   Sensorless mode (stCfg.bNoSensors): the TWELVE movement states ignore
   sensor feedback and advance when tStepTimeoutMs expires — the timeout
   doubles as the fixed step duration. Those twelve are both INIT_* sets
   (3), the three RECOVER_* states, both GRIP states and the four Sep/Push
   states. So error codes 1/3/4/5/6/7/8/10/11/12/13/14 are ALL unreachable
   while sensorless — this said "the 4 movement states" and "1/3/4/5",
   which was wrong before the RECOVER chain existed and is wronger now.
   CHECK_PLATE is deliberately NOT covered: it keeps its own
   tPlateWaitTimeoutMs and still needs a plate sensor, so error 9 stays
   reachable. Every bench run so far has had this flag set, which is why no
   movement-timeout path has ever been exercised on a panel. *)
VAR_INPUT
    (* External start pulse (rising-edge; one scan wide). MAIN fires this
       when the robot's CMD:1 arrives via TCP, or a physical PB1 rising
       edge in Auto mode. HMI START button and SimStartAssembly are
       consumed separately below via their own R_TRIGs. *)
    bExtStartPulse        : BOOL;

    (* Global machine-mode gate (GVL_HMI.bAutoMode). While FALSE the cycle is
       held in IDLE: every start trigger is ignored and a running cycle is
       aborted back to IDLE. This is the hard interlock that stops the
       operator or a stray robot edge starting motion while the machine is
       in Manual. *)
    bMachineAuto          : BOOL;

    (* BENCH SOAK FLAG -- log-file testing only. Wired by MAIN from
       GVL_HMI.bTempTestContinuesAutoRun, ticked online from the IDE. No HMI
       control by decision: an operator must not be able to reach it.

       While TRUE -- AND the build is a bench build, see bBenchBuild -- the
       machine self-arms out of NOT_HOMED and starts another bulb every time it
       reaches IDLE, with no operator START, no robot CMD:1 and no sim flag. So
       the log ring and the CSV fill continuously and rotation / retention can
       actually be exercised on a panel.

       LEVEL, not an edge, unlike every other term it is OR-ed into. That is the
       point: it has to re-fire on each arrival in IDLE.

       Three things it deliberately does NOT do, even on a bench build:
         - it does not bypass bMachineAuto, so Manual is still the hard stop;
         - it does not touch ERR, so a fault still ends the run (with bNoSensors
           AND bBypassPlateSensors set, no error code is reachable, so a soak
           should not fault at all -- if it does, that is a real finding);
         - it does not persist. GVL_HMI is plain VAR_GLOBAL, so the FALSE
           initialiser is re-applied on every cold boot and every download.

       NOTHING downstream reads this input directly. It is gated into
       bTempTestRun in Section 0a and every use site reads that. *)
    bTempTestContinuesAutoRun : BOOL;

    (* Per-pair sensor state. MAIN wires each element from stSepSolK/stPushSolK.bIs*. *)
    bSepIsExtended        : ARRAY[1..3] OF BOOL;
    bSepIsRetracted       : ARRAY[1..3] OF BOOL;
    bPushIsExtended       : ARRAY[1..3] OF BOOL;
    bPushIsRetracted      : ARRAY[1..3] OF BOOL;

    (* Grip pistons — L=[1], R=[2]. MAIN wires from stGripSolL/R.bIs*. *)
    bGripIsExtended       : ARRAY[1..2] OF BOOL;
    bGripIsRetracted      : ARRAY[1..2] OF BOOL;

    (* Plate-presence sensors gating CHECK_PLATE. Both must be TRUE before the
       cycle can advance out of CHECK_PLATE into GRIP_EXTENDING. Latched at
       cycle start only — not monitored past that step. *)
    bPlateSenL            : BOOL;
    bPlateSenR            : BOOL;
END_VAR

VAR_IN_OUT
    stHmi     : ST_HmiMasterAuto;
    stCfg     : ST_HmiMasterAutoCfg;
    stRobot   : ST_HmiRobot;
END_VAR

VAR_OUTPUT
    (* MAIN OR-merges these with the per-piston auto FBs. *)
    bSepCmdExtend         : ARRAY[1..3] OF BOOL;
    bSepCmdRetract        : ARRAY[1..3] OF BOOL;
    bPushCmdExtend        : ARRAY[1..3] OF BOOL;
    bPushCmdRetract       : ARRAY[1..3] OF BOOL;

    (* Grip piston commands. Extend held TRUE from GRIP_EXTENDING through
       SEP_RETRACTED_DWELL so the plate stays clamped for the entire cycle. *)
    bGripCmdExtend        : ARRAY[1..2] OF BOOL;
    bGripCmdRetract       : ARRAY[1..2] OF BOOL;

    (* TRUE while the master cycle is in any state other than IDLE or ERR.
       MAIN reads this to force enabled pistons' stHmi.eMode := Automatic
       while running, so bAutoCmd* actually reaches the piston coil (in
       Manual mode the piston FB ignores bAutoCmd*)
    bAnyRunning           : BOOL;
END_VAR

VAR
    (* Rising-edge detectors for momentary HMI buttons + robot start signal. *)
    fbTrigStart           : R_TRIG;
    fbTrigStop            : R_TRIG;
    fbTrigReset           : R_TRIG;
    fbTrigStartAssembly   : R_TRIG;
    fbTrigStartCycle      : R_TRIG;

    (* TEMPORARY -- mode-change log for the CSV soak-test flag. Delete with it. *)
    fbTrigTempTestOn      : R_TRIG;
    fbTrigTempTestOff     : F_TRIG;

    (* Rising-edge detectors for per-step Sim flags. *)
    fbSim_Idle            : R_TRIG;
    fbSim_InitPushRet     : R_TRIG;
    fbSim_InitSepRet      : R_TRIG;
    fbSim_InitGripRet     : R_TRIG;
    fbSim_WaitPlate       : R_TRIG;
    fbSim_GripExt         : R_TRIG;
    fbSim_SepExt          : R_TRIG;
    fbSim_PushExt         : R_TRIG;
    fbSim_DwellPush       : R_TRIG;
    fbSim_PushRet         : R_TRIG;
    fbSim_PushRetDwell    : R_TRIG;
    fbSim_SepRet          : R_TRIG;
    fbSim_SepRetDwell     : R_TRIG;
    fbSim_GripRet         : R_TRIG;
    fbSim_RecoverPushRet  : R_TRIG;
    fbSim_RecoverSepRet   : R_TRIG;
    fbSim_RecoverGripRet  : R_TRIG;

    (* Which exit the INIT retract chain takes when it completes:
         TRUE  -> IDLE         the chain was run to HOME the machine
                               (operator START, or recovery from ERR)
         FALSE -> CHECK_PLATE   the chain is the front of a bulb cycle
                               (robot CMD:1)
       Set by whoever ENTERS the chain, never from inside it -- the three INIT
       states are shared by both callers and must not care which one they serve. *)
    bHomeThenIdle         : BOOL;

    (* Per-step timer. Same TON, different PT depending on state. On DWELL
       states PT is the dwell; on wait states PT is the timeout. *)
    tonStep               : TON;

    (* Transition detect for the timer reset and the transition log. Seeded to
       NOT_HOMED to match stHmi.eStep's own default, so power-up does not log a
       phantom 'IDLE -> NOT_HOMED' for a state the machine was never in. *)
    ePrevStep             : E_MasterAutoStep := E_MasterAutoStep.NOT_HOMED;

    (* Loop index *)
    i                     : USINT;

    (* Aggregate sensor flags, computed each cycle in Section 1. *)
    bAllSepExtended       : BOOL;
    bAllSepRetracted      : BOOL;
    bAllPushExtended      : BOOL;
    bAllPushRetracted     : BOOL;
    bAllGripExtended      : BOOL;
    bAllGripRetracted     : BOOL;
    bPlateOk              : BOOL;

    (* Gated form of bTempTestContinuesAutoRun: the raw flag AND bBenchBuild.
       Every use site reads THIS and never the raw input, so the gate has exactly
       one application point and a future use site cannot forget it. *)
    bTempTestRun          : BOOL;
END_VAR

VAR CONSTANT
    (* BENCH-BUILD GATE for bTempTestContinuesAutoRun. FALSE in every build that
       goes on a production machine. Set TRUE only in an IDE session driving a
       bench panel, and set it back before the build that ships.

       Why a CONSTANT rather than another runtime flag: GVL_HMI carries
       TcHmiSymbol.AddSymbol, so everything in it is writable over ADS by
       FlowerPyHmi, by pb_test, or by any laptop with a route. "It is only ever
       set from the IDE" is a habit, not an interlock -- the same reasoning the
       CASE ELSE below applies to eStep. A VAR CONSTANT cannot be written at
       runtime by anything, so while this is FALSE the self-start path is
       provably unreachable no matter what lands in the GVL field.

       WHY THE PATH MUST NOT SHIP ENABLED. It starts a bulb without the robot's
       CMD:1, and CMD:1 is the ONLY guarantee the PLC has that the arm is clear
       of the stand: WAIT_POS2 was retired on exactly that basis (see the header
       note), so there is no independent check left. CHECK_PLATE is not a
       substitute -- plate-present says the plate was placed, not that the arm
       withdrew, and it is an OR on the one confirmed sensor, latched at entry.
       Second, it self-arms out of NOT_HOMED, which re-opens the Manual->Auto
       hazard the 2026-07-29 arming model closed: the START press after Manual is
       the operator confirming they are clear of the machine, and this skips it.
       Neither of those is fixed by the flag being volatile -- both are reachable
       inside a single power cycle. *)
    bBenchBuild : BOOL := FALSE;
END_VAR

(* ==========================================
   0a. RISING-EDGE DETECTORS
   ========================================== *)
fbTrigStart        (CLK := stHmi.bStart);
fbTrigStop         (CLK := stHmi.bStop);
fbTrigReset        (CLK := stHmi.bReset);
fbTrigStartAssembly(CLK := stHmi.bSimStartAssembly);
fbTrigStartCycle   (CLK := stHmi.bStartCycle);

(* Bench soak flag. THE GATE IS APPLIED HERE AND NOWHERE ELSE -- everything
   downstream reads bTempTestRun, so on a production build (bBenchBuild FALSE)
   it is FALSE whatever an ADS client writes to the GVL field.

   The two edge detectors deliberately watch the RAW flag, not the gated one, so
   that an attempt to enable it on a production build is still visible in the log
   instead of vanishing silently. *)
bTempTestRun := bBenchBuild AND bTempTestContinuesAutoRun;

fbTrigTempTestOn   (CLK := bTempTestContinuesAutoRun);
fbTrigTempTestOff  (CLK := bTempTestContinuesAutoRun);

fbSim_Idle        (CLK := stHmi.bSimStep_Idle);
fbSim_InitPushRet (CLK := stHmi.bSimStep_InitPushRet);
fbSim_InitSepRet  (CLK := stHmi.bSimStep_InitSepRet);
fbSim_InitGripRet (CLK := stHmi.bSimStep_InitGripRet);
fbSim_WaitPlate   (CLK := stHmi.bSimStep_WaitPlate);
fbSim_GripExt     (CLK := stHmi.bSimStep_GripExt);
fbSim_SepExt      (CLK := stHmi.bSimStep_SepExt);
fbSim_PushExt     (CLK := stHmi.bSimStep_PushExt);
fbSim_DwellPush   (CLK := stHmi.bSimStep_DwellPush);
fbSim_PushRet     (CLK := stHmi.bSimStep_PushRet);
fbSim_PushRetDwell(CLK := stHmi.bSimStep_PushRetDwell);
fbSim_SepRet      (CLK := stHmi.bSimStep_SepRet);
fbSim_SepRetDwell (CLK := stHmi.bSimStep_SepRetDwell);
fbSim_GripRet     (CLK := stHmi.bSimStep_GripRet);
fbSim_RecoverPushRet(CLK := stHmi.bSimStep_RecoverPushRet);
fbSim_RecoverSepRet (CLK := stHmi.bSimStep_RecoverSepRet);
fbSim_RecoverGripRet(CLK := stHmi.bSimStep_RecoverGripRet);

(* ==========================================
   0b. AUTO-CLEAR ONE-SHOT FLAGS ON RISING EDGE
   HMI button flags and Sim flags are momentary; after we detect the
   rising edge we clear the raw flag so the operator's next click can
   fire again. bExtStartPulse is already a one-scan pulse produced by
   MAIN's R_TRIG on the robot's TCP command channel -- nothing to clear.
   ========================================== *)
IF fbTrigStart.Q  THEN
    stHmi.bStart := FALSE;
    F_LogEvent(eSev := E_LogSev.INFO, sSource := stHmi.Name, sMsg := 'START pressed');
END_IF;
IF fbTrigStop.Q   THEN
    stHmi.bStop  := FALSE;
    F_LogEvent(eSev := E_LogSev.INFO, sSource := stHmi.Name, sMsg := 'STOP pressed');
END_IF;
IF fbTrigReset.Q  THEN
    stHmi.bReset := FALSE;
    F_LogEvent(eSev := E_LogSev.INFO, sSource := stHmi.Name, sMsg := 'RESET pressed');
END_IF;

(* Bench sim of the robot start: fires on the HMI checkbox rising edge and
   auto-clears. Log so bench-driven cycles show up in the event log. The
   robot-driven start comes in as bExtStartPulse (already an edge, no R_TRIG
   needed here) and is logged from MAIN when nRobotCmd goes 0->1. *)
IF fbTrigStartAssembly.Q THEN
    stHmi.bSimStartAssembly := FALSE;
    F_LogEvent(eSev := E_LogSev.INFO, sSource := stHmi.Name, sMsg := 'Sim start pressed');
END_IF;
(* Operator cycle start. Logged with its own message so the ring tells you
   WHO asked for the bulb: this, 'Sim start pressed' (bench stand-in for the
   robot), 'External start pulse' (the real robot, or the PB2+PB3 hold, both
   arriving as bExtStartPulse) and 'START pressed' (arming) are four
   different events and a fault report needs to tell them apart. *)
IF fbTrigStartCycle.Q THEN
    stHmi.bStartCycle := FALSE;
    F_LogEvent(eSev := E_LogSev.INFO, sSource := stHmi.Name,
               sMsg := 'Operator cycle start');
END_IF;
IF bExtStartPulse THEN
    F_LogEvent(eSev := E_LogSev.INFO, sSource := stHmi.Name, sMsg := 'External start pulse');
END_IF;

(* Bench soak flag, mode change. WARN on enable rather than INFO because a CSV
   read back weeks later has to say plainly that from this line onward the
   machine was self-running and every bulb below it is a test artefact, not
   production output.

   The refusal is logged too, and at WARN. On a production build the flag does
   nothing, and somebody who has just set it and is watching an idle machine
   needs to be told WHY rather than left to conclude the panel is broken -- this
   is the one line that says "rebuild with bBenchBuild TRUE". *)
IF fbTrigTempTestOn.Q THEN
    IF bBenchBuild THEN
        F_LogEvent(eSev := E_LogSev.WARN, sSource := stHmi.Name,
                   sMsg := 'BENCH SOAK continuous auto-run ENABLED');
    ELSE
        F_LogEvent(eSev := E_LogSev.WARN, sSource := stHmi.Name,
                   sMsg := 'Bench soak flag IGNORED - not a bench build');
    END_IF;
END_IF;
IF fbTrigTempTestOff.Q AND bBenchBuild THEN
    F_LogEvent(eSev := E_LogSev.INFO, sSource := stHmi.Name,
               sMsg := 'BENCH SOAK continuous auto-run disabled');
END_IF;

IF fbSim_Idle.Q         THEN stHmi.bSimStep_Idle         := FALSE; END_IF;
IF fbSim_InitPushRet.Q  THEN stHmi.bSimStep_InitPushRet  := FALSE; END_IF;
IF fbSim_InitSepRet.Q   THEN stHmi.bSimStep_InitSepRet   := FALSE; END_IF;
IF fbSim_InitGripRet.Q  THEN stHmi.bSimStep_InitGripRet  := FALSE; END_IF;
IF fbSim_WaitPlate.Q    THEN stHmi.bSimStep_WaitPlate    := FALSE; END_IF;
IF fbSim_GripExt.Q      THEN stHmi.bSimStep_GripExt      := FALSE; END_IF;
IF fbSim_SepExt.Q       THEN stHmi.bSimStep_SepExt       := FALSE; END_IF;
IF fbSim_PushExt.Q      THEN stHmi.bSimStep_PushExt      := FALSE; END_IF;
IF fbSim_DwellPush.Q    THEN stHmi.bSimStep_DwellPush    := FALSE; END_IF;
IF fbSim_PushRet.Q      THEN stHmi.bSimStep_PushRet      := FALSE; END_IF;
IF fbSim_PushRetDwell.Q THEN stHmi.bSimStep_PushRetDwell := FALSE; END_IF;
IF fbSim_SepRet.Q       THEN stHmi.bSimStep_SepRet       := FALSE; END_IF;
IF fbSim_SepRetDwell.Q  THEN stHmi.bSimStep_SepRetDwell  := FALSE; END_IF;
IF fbSim_GripRet.Q      THEN stHmi.bSimStep_GripRet      := FALSE; END_IF;

(* ==========================================
   1. AGGREGATE SENSOR STATE
   ========================================== *)
bAllSepExtended   := bSepIsExtended[1]   AND bSepIsExtended[2]   AND bSepIsExtended[3];
bAllSepRetracted  := bSepIsRetracted[1]  AND bSepIsRetracted[2]  AND bSepIsRetracted[3];
bAllPushExtended  := bPushIsExtended[1]  AND bPushIsExtended[2]  AND bPushIsExtended[3];
bAllPushRetracted := bPushIsRetracted[1] AND bPushIsRetracted[2] AND bPushIsRetracted[3];
bAllGripExtended  := bGripIsExtended[1]  OR bGripIsExtended[2];
bAllGripRetracted := bGripIsRetracted[1] OR bGripIsRetracted[2];
bPlateOk          := bPlateSenL OR bPlateSenR;

(* ==========================================
   2. GLOBAL OVERRIDES — STOP and RESET
   Both were rewritten 2026-07-29; this header used to describe the old
   behaviour ("STOP latches error 99 and drops to ERR, RESET returns to
   IDLE", plus a discrete-IO RESET_ALARM on robot DI 10 that no longer
   exists). What the three branches below actually do now:

     STOP   -> NOT_HOMED, error cleared. DISARMS, does not fault. Fires from
               IDLE too, giving the operator an explicit disarm.
     RESET  -> clears the error and enters the INIT homing chain with
               bHomeThenIdle TRUE. NOT straight to IDLE.
     Manual -> parks in NOT_HOMED (ERR stays latched), which is the whole
               implementation of "returning from Manual needs a START".

   RESET arrives either as the HMI button or as the robot's CMD:2, which MAIN
   fans into the same stHmi.bReset field — the robot resets the fault over
   TCP now, so there is nothing for the operator to reset on the robot side.
   ========================================== *)
IF fbTrigStop.Q AND stHmi.eStep <> E_MasterAutoStep.ERR THEN
    (* STOP DISARMS, it does not fault. Error code 99 ('Operator STOP while
       running') is retired.

       It used to latch ERR, which was harmless only while the CMD:1 latch bug
       masked it. Now that a re-sent command is honoured, ERR means the robot
       sees STATE:99, answers CMD:2, the PLC self-homes and reports IDLE, and
       the robot immediately starts another bulb -- i.e. a deliberate operator
       STOP would restart the machine within a couple of seconds.

       Dropping to NOT_HOMED instead reports 'wait' rather than 'fault', so the
       robot never tries to reset it, and the machine cannot move again until a
       human presses START. It also restores the distinction that ERR means
       something went WRONG, not that someone intervened.

       Fires from IDLE too, which gives the operator an explicit disarm: STOP in
       IDLE takes the machine out of the robot's reach. *)
    stHmi.iErrorCode := 0;
    stHmi.sErrorText := '';
    stHmi.eStep      := E_MasterAutoStep.NOT_HOMED;
END_IF;

IF fbTrigReset.Q AND stHmi.eStep = E_MasterAutoStep.ERR THEN
    (* RESET (operator button, or the robot's CMD:2 fanned in by MAIN) clears
       the fault and HOMES -- it does not drop straight to IDLE any more.

       Two reasons. A fault leaves the pistons in unknown positions, so going
       to IDLE would advertise STATE:0 ('ready') while the machine is not; and
       RESET landing in IDLE with the robot still asking for a bulb made RESET
       itself a start button, ~1 s after the operator cleared the fault. Now
       RESET only ever produces motion towards home, and the cycle starts on the
       robot's own CMD:1 once IDLE is genuinely reached. *)
    stHmi.iErrorCode := 0;
    stHmi.sErrorText := '';
    (* Recovery runs its OWN chain now, not the shared RETRACT/INIT one,
       so a failed recovery reports codes 12/13/14 and a distinct
       sStepText instead of looking exactly like a failed arming.
       bHomeThenIdle is irrelevant to that chain -- RECOVER_GRIP_RETR
       always exits to IDLE. *)
    stHmi.eStep      := E_MasterAutoStep.RECOVER_PUSH_RETR;
END_IF;

(* Global Auto/Manual hard interlock. Being in Manual forces the cycle out of
   any running state and drops Continuous, so a stray robot start pulse cannot
   restart motion. Not treated as a fault (no ERR/error code) — Manual is a
   normal operator choice, not an alarm. ERR stays latched until RESET.

   Parks in NOT_HOMED rather than IDLE, and THAT is the whole implementation of
   "returning from Manual needs an operator START": manual jogging can leave the
   pistons anywhere, so the machine must be un-armed when Auto comes back. No
   Manual->Auto edge detection is needed — the state is simply already
   NOT_HOMED, and the operator's START homes it. *)
IF NOT bMachineAuto AND stHmi.eStep <> E_MasterAutoStep.NOT_HOMED AND stHmi.eStep <> E_MasterAutoStep.ERR THEN
    stHmi.eStep       := E_MasterAutoStep.NOT_HOMED;
END_IF;

(* ==========================================
   3. STEP TIMER + TRANSITION LOG
   Reset tonStep on any state change. In DWELL states PT is the dwell
   duration and Q rising = "dwell complete, advance". In wait states PT
   is the timeout and Q rising = "timed out, error". Non-waiting states
   (IDLE, ERR) do not consult Q.

   Also emit one log entry per transition — INFO with "PREV -> NEW" for
   normal advances, ERR with sErrorText when the new state is ERR. The
   check runs one scan AFTER Section 4 set eStep, so sErrorText and
   iErrorCode are already populated. Order matters: log BEFORE updating
   ePrevStep so both endpoints are still available.
   ========================================== *)
IF stHmi.eStep <> ePrevStep THEN
    IF stHmi.eStep = E_MasterAutoStep.ERR THEN
        F_LogEvent(eSev := E_LogSev.ERR, sSource := stHmi.Name, sMsg := stHmi.sErrorText);
    ELSE
        F_LogEvent(
            eSev    := E_LogSev.INFO,
            sSource := stHmi.Name,
            sMsg    := CONCAT(CONCAT(TO_STRING(ePrevStep), ' -> '), TO_STRING(stHmi.eStep))
        );
    END_IF

    tonStep(IN := FALSE, PT := T#0MS);   // pulse-off resets ET to 0
    ePrevStep := stHmi.eStep;
END_IF;

(* PT depends on state. Wait states use tStepTimeoutMs; dwell states use their own.
   CHECK_PLATE uses tPlateWaitTimeoutMs (bounded by robot placement time). *)
CASE stHmi.eStep OF
    E_MasterAutoStep.DWELL_PUSH:
        tonStep(IN := TRUE, PT := UDINT_TO_TIME(stCfg.tDwellPushMs));
    E_MasterAutoStep.PUSH_RETRACTED_DWELL:
        tonStep(IN := TRUE, PT := UDINT_TO_TIME(stCfg.tPushRetractedDwellMs));
    E_MasterAutoStep.SEP_RETRACTED_DWELL:
        tonStep(IN := TRUE, PT := UDINT_TO_TIME(stCfg.tSepRetractedDwellMs));
    E_MasterAutoStep.CHECK_PLATE:
        tonStep(IN := TRUE, PT := UDINT_TO_TIME(stCfg.tPlateWaitTimeoutMs));
    E_MasterAutoStep.SEP_EXTENDING,
    E_MasterAutoStep.PUSH_EXTENDING,
    E_MasterAutoStep.PUSH_RETRACTING,
    E_MasterAutoStep.SEP_RETRACTING,
    E_MasterAutoStep.INIT_PUSH_RETRACTING,
    E_MasterAutoStep.INIT_SEP_RETRACTING,
    E_MasterAutoStep.INIT_GRIP_RETRACTING,
    E_MasterAutoStep.GRIP_EXTENDING,
    E_MasterAutoStep.GRIP_RETRACTING,
    E_MasterAutoStep.RECOVER_PUSH_RETR,
    E_MasterAutoStep.RECOVER_SEP_RETR,
    E_MasterAutoStep.RECOVER_GRIP_RETR:
        tonStep(IN := TRUE, PT := UDINT_TO_TIME(stCfg.tStepTimeoutMs));
ELSE
    tonStep(IN := FALSE, PT := T#0MS);
END_CASE;

stHmi.tElapsedS := DINT_TO_LREAL(TIME_TO_DINT(tonStep.ET)) / 1000.0;

(* ==========================================
   4. STATE MACHINE
   Default: clear all commands each cycle in the ELSE-ish paths so a
   dropped state doesn't leave stale coils driven. Each state re-asserts
   the commands it owns. Grip commands are held TRUE from GRIP_EXTENDING
   through SEP_RETRACTED_DWELL so the plate stays clamped for the entire
   Sep/Push cycle.
   ========================================== *)
CASE stHmi.eStep OF

    E_MasterAutoStep.IDLE:
        ResetAllCommands();
        (* No active error while in IDLE (unless just about to enter ERR
           via a global override, handled above). *)
        stHmi.iErrorCode := 0;
        stHmi.sErrorText := '';

        (* ONLY THE ROBOT STARTS A BULB CYCLE.

           fbTrigStart.Q (operator START) and the retired stCfg.bContinuous were
           removed from this condition. That is the point of the whole arming
           model: START means "home and arm", and Continuous would re-arm with
           nothing external gating it at all. What is left is the robot's CMD:1
           (arriving as bExtStartPulse -- which is also how the PB2+PB3 hold
           arrives), the operator's own bStartCycle, its bench stand-in
           bSimStartAssembly, and the per-step sim flag.

           bStartCycle is a SEPARATE field from bStart on purpose, and the
           distinction is the whole reason START was removed from here: bStart
           means "home and arm" in NOT_HOMED, so overloading it to also mean
           "run a bulb" in IDLE would restore the two-meanings-one-symbol
           problem that let a green-before-orange combo press lose its
           request. A separate command cannot be misread by state.

           Still gated by bMachineAuto: in Manual nothing starts, even on a
           robot pulse (no double-control).

           Enters the INIT chain rather than CHECK_PLATE directly so pistons left
           somewhere unexpected are driven home first; with everything already
           retracted the three INIT states self-satisfy on the next scan, so it
           costs nothing per bulb. bHomeThenIdle FALSE routes the chain's exit
           on to CHECK_PLATE and the rest of the cycle. *)
        (* bTempTestRun is OR-ed in as a LEVEL, so the moment the machine lands
           back in IDLE it starts the next bulb -- that is what makes a soak
           self-sustaining. Compile-time FALSE unless bBenchBuild is set, so this
           term does not exist on a production build. *)
        IF bMachineAuto AND (bExtStartPulse OR fbTrigStartCycle.Q
                             OR fbTrigStartAssembly.Q OR fbSim_Idle.Q
                             OR bTempTestRun) THEN
            (* Logged per cycle, not just once when the flag goes TRUE, because
               aRecent is only 20 slots deep -- the enable WARN scrolls out of
               the panel ring within two bulbs, and without this line the Logs
               page would show bulb after bulb with nothing saying what started
               them. In the CSV it is redundant with the WARN; on the panel it is
               the only answer.

               Gated, not raw: on a production build a genuine robot-started bulb
               must not be labelled a soak cycle just because someone set the GVL
               field over ADS. *)
            IF bTempTestRun THEN
                F_LogEvent(eSev := E_LogSev.INFO, sSource := stHmi.Name,
                           sMsg := 'BENCH SOAK auto-run cycle start');
            END_IF;
            bHomeThenIdle := FALSE;
            stHmi.eStep   := E_MasterAutoStep.INIT_PUSH_RETRACTING;
        END_IF;

        (* OPERATOR START IS IGNORED HERE (2026-08-05). It used to re-home and
           come back, justified as "harmless, and it keeps START's meaning
           identical in every state". Removed for two reasons.

           It was a no-op in outcome. Nothing can disturb a piston while we sit
           in IDLE: each valve output has exactly one writer -- its piston FB's
           bOutSolenoid -- and in Automatic the auto commands are all FALSE here,
           the HMI Extend/Retract selections are force-cleared every scan, and
           the PB jogs are not available in any Auto state. IDLE is only reached
           from INIT_GRIP_RETRACTING, GRIP_RETRACTING or RECOVER_GRIP_RETR, all
           of which end with everything retracted. So the pistons were already
           home and the INIT chain self-satisfied.

           And it cost a real defect. Because the re-home left IDLE, an operator
           pressing GREEN before ORANGE for the PB2+PB3 bulb-start combo could
           have the combo's one-scan bExtStartPulse land while eStep was still in
           the INIT chain -- where nothing consumes it -- so the request was
           silently dropped and no bulb ran. Measured on the machine. With START
           ignored here the machine never leaves IDLE, so that pulse always lands
           somewhere that consumes it. This removes the cause rather than
           tolerating it.

           The position-proof the re-home offered is still reachable, just
           deliberately: STOP (red PB held) drops to NOT_HOMED, and START from
           there homes and re-arms.

           fbTrigStart.Q is still consumed by Section 0b -- it is cleared and
           logged as 'START pressed' -- so a press here is visible in the log
           and simply has no effect, exactly like a press during a cycle. *)

    E_MasterAutoStep.NOT_HOMED:
        (* In Automatic but NOT armed: entered on power-up (stHmi.eStep's
           declared default), on any time spent in Manual, and on operator STOP.
           nStateOut reports 40, which the robot treats as "wait" -- it is
           neither IDLE(0) "send me a bulb" nor ERR(99) "reset me".

           Nothing is driven and no timer runs (Section 3 falls to its ELSE, as
           for IDLE). The ONLY exit is an operator START -- the HMI button or the
           green PB3, which MAIN maps onto the same stHmi.bStart field. *)
        ResetAllCommands();

        stHmi.iErrorCode := 0;
        stHmi.sErrorText := '';

        (* bTempTestRun self-arms, so a soak needs no operator START at all: tick
           the flag online and the machine homes and then cycles.

           THIS IS THE TERM THAT MAKES THE GATE NECESSARY. Skipping the START
           press also skips the operator confirming they are clear of the
           machine, so on a Manual -> Auto return it re-opens the hazard the
           arming model closed. Compile-time FALSE unless bBenchBuild is set.

           No log line here: this fires once per enable, and the enable WARN is
           the entry immediately before it with Section 3's
           NOT_HOMED -> INIT_PUSH_RETRACTING right after. *)
        IF bMachineAuto AND (fbTrigStart.Q OR bTempTestRun) THEN
            bHomeThenIdle := TRUE;
            stHmi.eStep   := E_MasterAutoStep.INIT_PUSH_RETRACTING;
        END_IF;

    E_MasterAutoStep.INIT_PUSH_RETRACTING:
        (* Mirror end-of-cycle PUSH_RETRACTING: assert push retract only. Sep
           stays uncommanded (whatever position it was left in — its retract
           follows in INIT_SEP_RETRACTING). Grip uncommanded here. *)
        ResetAllCommands();
        FOR i := 1 TO 3 DO
            bPushCmdRetract[i] := TRUE;
        END_FOR;

        IF bAllPushRetracted OR fbSim_InitPushRet.Q OR (stCfg.bNoSensors AND tonStep.Q) THEN
            stHmi.eStep := E_MasterAutoStep.INIT_SEP_RETRACTING;
        ELSIF tonStep.Q THEN
            stHmi.iErrorCode := 6;
            stHmi.sErrorText := 'INIT_PUSH_RETRACTING timed out';
            stHmi.eStep := E_MasterAutoStep.ERR;
        END_IF;

    E_MasterAutoStep.INIT_SEP_RETRACTING:
        (* Push is confirmed home; now retract sep. *)
        ResetAllCommands();
        FOR i := 1 TO 3 DO
            bSepCmdRetract[i] := TRUE;
        END_FOR;

        IF bAllSepRetracted OR fbSim_InitSepRet.Q OR (stCfg.bNoSensors AND tonStep.Q) THEN
            stHmi.eStep := E_MasterAutoStep.INIT_GRIP_RETRACTING;
        ELSIF tonStep.Q THEN
            stHmi.iErrorCode := 7;
            stHmi.sErrorText := 'INIT_SEP_RETRACTING timed out';
            stHmi.eStep := E_MasterAutoStep.ERR;
        END_IF;

    E_MasterAutoStep.INIT_GRIP_RETRACTING:
        (* Both Sep and Push confirmed home; now retract grip. Defensive
           symmetry with INIT_PUSH_RETRACTING / INIT_SEP_RETRACTING so a
           prior manual jog does not leave grip clamped when the plate
           arrives. *)
        ResetAllCommands();
        FOR i := 1 TO 2 DO
            bGripCmdRetract[i] := TRUE;
        END_FOR;

        IF bAllGripRetracted OR fbSim_InitGripRet.Q OR (stCfg.bNoSensors AND tonStep.Q) THEN
            (* End of the shared retract chain -- the one place the two callers
               diverge. Homing (operator START, or ERR recovery) stops here with
               the machine armed; a robot-started cycle carries on into the bulb
               sequence. Everything above this line is identical for both. *)
            IF bHomeThenIdle THEN
                stHmi.eStep := E_MasterAutoStep.IDLE;
            ELSE
                stHmi.eStep := E_MasterAutoStep.CHECK_PLATE;
            END_IF;
        ELSIF tonStep.Q THEN
            stHmi.iErrorCode := 8;
            stHmi.sErrorText := 'INIT_GRIP_RETRACTING timed out';
            stHmi.eStep := E_MasterAutoStep.ERR;
        END_IF;

    E_MasterAutoStep.CHECK_PLATE:
        (* Nothing driven — waiting for the robot to place the plate on the
           fixture. Both plate sensors must confirm TRUE before advancing.
           No sensorless fallback: the whole point of this state is to gate
           on the plate presence. Timeout uses tPlateWaitTimeoutMs (see
           Section 3 timer selector). *)
        ResetAllCommands();

        IF bPlateOk OR fbSim_WaitPlate.Q THEN
            stHmi.eStep := E_MasterAutoStep.GRIP_EXTENDING;
        ELSIF tonStep.Q THEN
            (* Bypass removes only the ERROR, not the wait. The sensor
               fast-path above still applies, so with working sensors the
               cycle is unchanged; with unwired or faulty ones
               tPlateWaitTimeoutMs degrades into a fixed placement dwell and
               we carry on. That mirrors how bNoSensors turns tStepTimeoutMs
               into a fixed step duration, and it keeps the plate gate honest
               by default -- bNoSensors deliberately does NOT skip this
               state, so bypassing it has to be an explicit, separate
               decision. *)
            IF stCfg.bBypassPlateSensors THEN
                stHmi.eStep := E_MasterAutoStep.GRIP_EXTENDING;
            ELSE
                stHmi.iErrorCode := 9;
                stHmi.sErrorText := 'CHECK_PLATE timed out (plate never arrived)';
                stHmi.eStep := E_MasterAutoStep.ERR;
            END_IF;
        END_IF;

    E_MasterAutoStep.GRIP_EXTENDING:
        (* Plate is on the fixture; clamp it from both sides. *)
        ResetAllCommands();
        FOR i := 1 TO 2 DO
            bGripCmdExtend[i] := TRUE;
        END_FOR;

        IF bAllGripExtended OR fbSim_GripExt.Q OR (stCfg.bNoSensors AND tonStep.Q) THEN
            stHmi.eStep := E_MasterAutoStep.SEP_EXTENDING;
        ELSIF tonStep.Q THEN
            stHmi.iErrorCode := 10;
            stHmi.sErrorText := 'GRIP_EXTENDING timed out';
            stHmi.eStep := E_MasterAutoStep.ERR;
        END_IF;

    E_MasterAutoStep.SEP_EXTENDING:
        ResetAllCommands();
        FOR i := 1 TO 3 DO
            bSepCmdExtend[i] := TRUE;
        END_FOR;
        FOR i := 1 TO 2 DO
            bGripCmdExtend[i] := TRUE;   (* hold grip clamped *)
        END_FOR;

        IF bAllSepExtended OR fbSim_SepExt.Q OR (stCfg.bNoSensors AND tonStep.Q) THEN
            (* Skip the former WAIT_POS2 — the robot has already moved clear
               of the stand before signaling start via TCP CMD:1. *)
            stHmi.eStep := E_MasterAutoStep.PUSH_EXTENDING;
        ELSIF tonStep.Q THEN   (* only reachable when NOT bNoSensors *)
            stHmi.iErrorCode := 1;
            stHmi.sErrorText := 'SEP_EXTENDING timed out';
            stHmi.eStep := E_MasterAutoStep.ERR;
        END_IF;

    E_MasterAutoStep.PUSH_EXTENDING:
        ResetAllCommands();
        FOR i := 1 TO 3 DO
            bSepCmdExtend[i]  := TRUE;   (* hold sep out *)
            bPushCmdExtend[i] := TRUE;
        END_FOR;
        FOR i := 1 TO 2 DO
            bGripCmdExtend[i] := TRUE;
        END_FOR;

        IF bAllPushExtended OR fbSim_PushExt.Q OR (stCfg.bNoSensors AND tonStep.Q) THEN
            stHmi.eStep := E_MasterAutoStep.DWELL_PUSH;
        ELSIF tonStep.Q THEN
            stHmi.iErrorCode := 3;
            stHmi.sErrorText := 'PUSH_EXTENDING timed out';
            stHmi.eStep := E_MasterAutoStep.ERR;
        END_IF;

    E_MasterAutoStep.DWELL_PUSH:
        (* Hold everything out. *)
        ResetAllCommands();
        FOR i := 1 TO 3 DO
            bSepCmdExtend[i]  := TRUE;
            bPushCmdExtend[i] := TRUE;
        END_FOR;
        FOR i := 1 TO 2 DO
            bGripCmdExtend[i] := TRUE;
        END_FOR;

        IF tonStep.Q OR fbSim_DwellPush.Q THEN
            stHmi.eStep := E_MasterAutoStep.PUSH_RETRACTING;
        END_IF;

    E_MasterAutoStep.PUSH_RETRACTING:
        (* Sep still extended, push retract command asserted. *)
        ResetAllCommands();
        FOR i := 1 TO 3 DO
            bSepCmdExtend[i]   := TRUE;
            bPushCmdRetract[i] := TRUE;
        END_FOR;
        FOR i := 1 TO 2 DO
            bGripCmdExtend[i] := TRUE;
        END_FOR;

        IF bAllPushRetracted OR fbSim_PushRet.Q OR (stCfg.bNoSensors AND tonStep.Q) THEN
            stHmi.eStep := E_MasterAutoStep.PUSH_RETRACTED_DWELL;
        ELSIF tonStep.Q THEN
            stHmi.iErrorCode := 4;
            stHmi.sErrorText := 'PUSH_RETRACTING timed out';
            stHmi.eStep := E_MasterAutoStep.ERR;
        END_IF;

    E_MasterAutoStep.PUSH_RETRACTED_DWELL:
        (* Sep still held extended, push commands cleared. *)
        ResetAllCommands();
        FOR i := 1 TO 3 DO
            bSepCmdExtend[i] := TRUE;
        END_FOR;
        FOR i := 1 TO 2 DO
            bGripCmdExtend[i] := TRUE;
        END_FOR;

        IF tonStep.Q OR fbSim_PushRetDwell.Q THEN
            stHmi.eStep := E_MasterAutoStep.SEP_RETRACTING;
        END_IF;

    E_MasterAutoStep.SEP_RETRACTING:
        ResetAllCommands();
        FOR i := 1 TO 3 DO
            bSepCmdRetract[i] := TRUE;
        END_FOR;
        FOR i := 1 TO 2 DO
            bGripCmdExtend[i] := TRUE;
        END_FOR;

        IF bAllSepRetracted OR fbSim_SepRet.Q OR (stCfg.bNoSensors AND tonStep.Q) THEN
            stHmi.eStep := E_MasterAutoStep.SEP_RETRACTED_DWELL;
        ELSIF tonStep.Q THEN
            stHmi.iErrorCode := 5;
            stHmi.sErrorText := 'SEP_RETRACTING timed out';
            stHmi.eStep := E_MasterAutoStep.ERR;
        END_IF;

    E_MasterAutoStep.SEP_RETRACTED_DWELL:
        (* Sep/Push home; grip still clamped (released in GRIP_RETRACTING). *)
        ResetAllCommands();
        FOR i := 1 TO 2 DO
            bGripCmdExtend[i] := TRUE;
        END_FOR;

        IF tonStep.Q OR fbSim_SepRetDwell.Q THEN
            stHmi.eStep := E_MasterAutoStep.GRIP_RETRACTING;
        END_IF;

    E_MasterAutoStep.GRIP_RETRACTING:
        (* Very last motion: release the plate. On successful retract,
           increment nCyclesCompleted and return to IDLE. *)
        ResetAllCommands();
        FOR i := 1 TO 2 DO
            bGripCmdRetract[i] := TRUE;
        END_FOR;

        IF bAllGripRetracted OR fbSim_GripRet.Q OR (stCfg.bNoSensors AND tonStep.Q) THEN
            stHmi.nCyclesCompleted := stHmi.nCyclesCompleted + 1;
            (* Back to IDLE -- still ARMED, so the robot's next CMD:1 (or an
               operator START) runs the next bulb. Nothing re-arms by itself. *)
            stHmi.eStep := E_MasterAutoStep.IDLE;
        ELSIF tonStep.Q THEN
            stHmi.iErrorCode := 11;
            stHmi.sErrorText := 'GRIP_RETRACTING timed out';
            stHmi.eStep := E_MasterAutoStep.ERR;
        END_IF;

    (* ---- FAULT-RECOVERY RETRACT CHAIN (2026-08-05) ------------------
       Same motion and the same collision ordering as the RETRACT/INIT
       chain -- push, then sep, then grip -- but with its own identity, so
       the panel, the log and the wire can all tell a failed RECOVERY from
       a failed ARMING. Entered only from ERR on RESET; always exits to
       IDLE, because at that point the machine really is homed.
       ----------------------------------------------------------------- *)
    E_MasterAutoStep.RECOVER_PUSH_RETR:
        ResetAllCommands();
        FOR i := 1 TO 3 DO
            bPushCmdRetract[i] := TRUE;
        END_FOR;

        IF bAllPushRetracted OR fbSim_RecoverPushRet.Q OR (stCfg.bNoSensors AND tonStep.Q) THEN
            stHmi.eStep := E_MasterAutoStep.RECOVER_SEP_RETR;
        ELSIF tonStep.Q THEN
            stHmi.iErrorCode := 12;
            stHmi.sErrorText := 'RECOVER push retract timed out';
            stHmi.eStep := E_MasterAutoStep.ERR;
        END_IF;

    E_MasterAutoStep.RECOVER_SEP_RETR:
        ResetAllCommands();
        FOR i := 1 TO 3 DO
            bSepCmdRetract[i] := TRUE;
        END_FOR;

        IF bAllSepRetracted OR fbSim_RecoverSepRet.Q OR (stCfg.bNoSensors AND tonStep.Q) THEN
            stHmi.eStep := E_MasterAutoStep.RECOVER_GRIP_RETR;
        ELSIF tonStep.Q THEN
            stHmi.iErrorCode := 13;
            stHmi.sErrorText := 'RECOVER sep retract timed out';
            stHmi.eStep := E_MasterAutoStep.ERR;
        END_IF;

    E_MasterAutoStep.RECOVER_GRIP_RETR:
        ResetAllCommands();
        FOR i := 1 TO 2 DO
            bGripCmdRetract[i] := TRUE;
        END_FOR;

        IF bAllGripRetracted OR fbSim_RecoverGripRet.Q OR (stCfg.bNoSensors AND tonStep.Q) THEN
            stHmi.eStep := E_MasterAutoStep.IDLE;
        ELSIF tonStep.Q THEN
            stHmi.iErrorCode := 14;
            stHmi.sErrorText := 'RECOVER grip retract timed out';
            stHmi.eStep := E_MasterAutoStep.ERR;
        END_IF;

    E_MasterAutoStep.ERR:
        (* Latched. nStateOut mirrors ERR(99) so the robot's TCP client
           sees the fault via STATE:99 and can invoke its own error
           handler. Exit only via Section 2 (HMI RESET or CMD:2). *)
        ResetAllCommands();

ELSE
    (* Defensive: any eStep with no branch above lands here, and it snaps to
       NOT_HOMED -- NOT IDLE. IDLE is wire value 0, the one value that makes
       the robot send CMD:1, and this path is reached with the pistons in
       unknown positions. It is genuinely reachable: GVL_HMI carries
       TcHmiSymbol.AddSymbol so eStep is writable over ADS, and WAIT_POS2(2)
       is a declared enumerator with no branch. NOT_HOMED reports 'wait' and
       requires a human START. *)
    ResetAllCommands();
    stHmi.eStep := E_MasterAutoStep.NOT_HOMED;
END_CASE;

(* ==========================================
   5. STATUS MIRROR — human-readable step name + running flag
   TO_STRING relies on the enum's {to_string} attribute.
   bAnyRunning is TRUE any time the cycle is actively driving pistons —
   MAIN uses it to force enabled pistons into Automatic mode. False in ERR
   so the operator's manual choice is preserved after a fault.

   The "PLC is running" signal to the robot is derived robot-side from
   nStateOut != IDLE (see FB_RobotTcpClient); no separate outbound field
   needed here.
   ========================================== *)
stHmi.sStepText := TO_STRING(stHmi.eStep);
bAnyRunning     := (stHmi.eStep <> E_MasterAutoStep.IDLE)
               AND (stHmi.eStep <> E_MasterAutoStep.ERR);

(* Drive every piston command FALSE.

   Called at the top of EVERY state in Section 4, which then re-asserts only
   the commands it actually owns. That replaces the previous mix of explicit
   clears and commands held by omission -- eight of sixteen states cleared
   the full set and the rest inherited FALSE from whichever state ran before,
   so reading one branch in isolation could not tell you what the coils were
   doing.

   Behaviour is unchanged: each old body's net effect was already
   'everything FALSE except the commands it listed'. This makes that
   explicit, and makes a forgotten clear impossible.

   NOTE it clears COMMANDS, not coils. FB_SolSpringPiston_2Pos RETAINS its
   coil when no command branch matches, so clearing commands mid-stroke holds
   the piston where it is rather than dropping it. That is exactly why every
   state has to re-assert what it wants, every scan.

   Uses its own loop counter -- the FB's `i` belongs to the caller. *)
METHOD ResetAllCommands
VAR
    k : INT;
END_VAR
FOR k := 1 TO 3 DO
    bSepCmdExtend[k]   := FALSE;
    bSepCmdRetract[k]  := FALSE;
    bPushCmdExtend[k]  := FALSE;
    bPushCmdRetract[k] := FALSE;
END_FOR;
FOR k := 1 TO 2 DO
    bGripCmdExtend[k]  := FALSE;
    bGripCmdRetract[k] := FALSE;
END_FOR;
END_METHOD

END_FUNCTION_BLOCK

// ---- POUs/F_LogEvent.TcPOU
(*
    Push one entry into the GVL_Log ring buffer.

    Callable from any scan without side effects on control logic. DEBUG entries
    are dropped when GVL_Log.bDebugMode = FALSE, so leaving DBG calls in
    production code costs nothing.

    Returns TRUE if the entry was recorded, FALSE if dropped by the debug filter.
*)
FUNCTION F_LogEvent : BOOL
VAR_INPUT
    eSev    : E_LogSev;
    sSource : STRING(20);
    sMsg    : STRING(80);
END_VAR
VAR
    idx : UDINT;
    k   : INT;
END_VAR

// Global mute — operator can disable ALL PLC logging from the HMI. When
// FALSE, we drop the event silently; the ring buffer and aRecent mirror
// are not touched so the last-known state stays visible.
IF NOT GVL_Log.bLogEnabled THEN
    F_LogEvent := FALSE;
    RETURN;
END_IF

// Debug filter — drop DBG severity when debug mode is off
IF (eSev = E_LogSev.DBG) AND NOT GVL_Log.bDebugMode THEN
    F_LogEvent := FALSE;
    RETURN;
END_IF

// Write into the ring at slot = nWriteIdx MOD 256
idx := GVL_Log.nWriteIdx MOD 256;
GVL_Log.aLog[idx].eSev     := eSev;
GVL_Log.aLog[idx].sSevText := TO_STRING(eSev);
GVL_Log.aLog[idx].sTime    := GVL_Log.sNow;
GVL_Log.aLog[idx].sSource  := sSource;
GVL_Log.aLog[idx].sMsg     := sMsg;

// Shift the newest-first mirror down by one and write the new entry at
// [0]. HMI Logs page binds aRecent[0..19] directly in display order.
// The shift copies whole structs, so sSevText rides along with no extra work.
FOR k := 19 TO 1 BY -1 DO
    GVL_Log.aRecent[k] := GVL_Log.aRecent[k-1];
END_FOR
GVL_Log.aRecent[0].eSev     := eSev;
GVL_Log.aRecent[0].sSevText := TO_STRING(eSev);
GVL_Log.aRecent[0].sTime    := GVL_Log.sNow;
GVL_Log.aRecent[0].sSource  := sSource;
GVL_Log.aRecent[0].sMsg     := sMsg;

// Increment the monotonic write counter — Python bridge polls this and
// drains any slots between its lastReadIdx and this value.
GVL_Log.nWriteIdx := GVL_Log.nWriteIdx + 1;

F_LogEvent := TRUE;

END_FUNCTION

// ---- POUs/FB_RobotTcpClient.TcPOU
(*
   TCP/IP client for the Dobot protocol on port 6001. Robot is the TCP
   server; PLC dials in. Robot comms are TCP-ONLY: the former discrete-I/O
   handshake (STAND_SEQ_DO / STAND_SEQ_DI) is retired and its channels
   (DI[13], DO[7]) are now free. Uses the free-with-TF6310 Tc2_TcpIp
   socket FBs; empty sSrvNetId targets the local TwinCAT TCP/IP Connection
   Server.

   Protocol (raw ASCII, no newline framing; one send -> one reply, matching
   RobotBridge\Client_working_example\tcp client.py / dummy_server.py):
     PLC -> robot        robot -> PLC
     "GET_SYNC"          "SYNC:J_SPEED=10,L_SPEED=10,..."
     "NAME:VALUE"        "OK: SET NAME"
     "New_Bulb:1"        "OK: SET New_Bulb"
     "STATE:n"           "CMD:m"

   STATE frames are the PLC's continuous state push (n = INT value of
   E_MasterAutoStep, or MANUAL=30 when bAutoMode=FALSE). Sent on every
   change of stParams.nStateOut and every IDLE_STATE_MS as keep-alive.
   The robot's reply carries the next command (m in {0,1,2}: 0=none,
   1=start cycle, 2=reset error) which ParseCmd writes to
   stParams.nRobotCmd. MAIN consumes that field as a level and clears it.

   Tuning params are bidirectional. GET_SYNC pulls all 11 into stParams
   after every connect, and the FB then snapshots them into aShadow. Any
   later divergence between a live field and its shadow slot is treated as
   an operator edit and pushed back as NAME:VALUE, one param per
   round-trip. So an HMI NumericInput can bind straight to
   GVL_Robot.stParams.J_SPEED and simply work -- no request flags to set.
   The bSetParam / sSetName / nSetVal triple remains as a raw escape hatch
   for names that are not struct fields.

   Known limitation: stParams is both setpoint and actual. An edit made
   while the link is down is overwritten by the GET_SYNC that follows the
   next reconnect. Separating desired-vs-actual would need a second struct.

   State machine mirrors the Python supervisor: Disconnected -> Connecting
   -> Connected; any socket error closes and re-dials after RECONNECT_MS.
*)
FUNCTION_BLOCK FB_RobotTcpClient
VAR_INPUT
    // Master enable. FALSE tears down any connection and holds Disconnected.
    bEnable     : BOOL;
    // Robot server target (from GVL_Robot.sRobotHost / nRobotPort).
    sRemoteHost : STRING;
    nRemotePort : UINT;
END_VAR
VAR_IN_OUT
    // Status mirror for the HMI (eConnState, packet counts, last messages).
    stRobot  : ST_HmiRobot;
    // Tuning params + request flags; SYNC replies parse back into this.
    stParams : ST_RobotParams;
END_VAR
VAR
    fbConnect : FB_SocketConnect;
    fbClose   : FB_SocketClose;
    fbSend    : FB_SocketSend;
    fbReceive : FB_SocketReceive;
    hSocket   : T_HSOCKET;

    // Empty => local TwinCAT TCP/IP Connection Server (TF6310).
    sSrvNetId : T_AmsNetId := '';

    eState : E_RobotConnState := E_RobotConnState.Disconnected;
    iIo    : INT;            // request/reply sub-state while Connected
    iPend  : INT;            // which message we last sent (drives reply parse)

    tonReconnect : TON;      // delay before re-dial after a drop
    tonIdle      : TON;      // idle -> STATE keep-alive
    tonReply     : TON;      // reply timeout guard

    sTxMsg    : STRING(255);
    sRxMsg    : STRING(255);
    aRxBuffer : ARRAY[0..255] OF BYTE;

    bAutoSyncQueued : BOOL;  // one-shot GET_SYNC right after each (re)connect
    nLastStateSent  : INT := -1;   // last nStateOut we transmitted; -1 forces first push

    // Shadow copy of the 11 tuning params, used to detect operator edits.
    // Snapshotted from stParams after every GET_SYNC round-trip; any later
    // divergence means "the HMI changed this field" and is pushed to the
    // robot as NAME:VALUE. Held invalid until the first SYNC completes so
    // the power-on defaults are never mistaken for edits.
    aShadow      : ARRAY[1..11] OF INT;
    bShadowValid : BOOL;

    // Which param the in-flight TX_SETPARAM belongs to. 0 = the explicit
    // bSetParam/sSetName/nSetVal escape hatch (no shadow slot to update).
    nPendIdx : INT;
    nPendVal : INT;   // value actually sent; written to aShadow on ACK
END_VAR
VAR
    // ------------------------------- LOGGING (see the Fail method for policy)
    // Every robot event is pushed into GVL_Log through F_LogEvent, so the panel
    // Logs page and FlowerPyHmi both see it. Lifecycle and protocol events log
    // at INFO / WARN / ERR; raw frames log at DBG, which F_LogEvent drops
    // unless GVL_Log.bDebugMode is set. So production stays readable and
    // ticking Debug turns this FB into a protocol tracer.
    //
    // The ring is only 20 entries deep on the panel page, which is why the two
    // repeating events below are edge-logged rather than level-logged.

    // Last CMD value logged. The robot may repeat a command across several
    // replies before zeroing it, so commands log on change only. Baselined
    // even for CMD:0, so the next non-zero value is not read as a repeat.
    nLastCmdLogged : INT;

    // TRUE while STATE pushes are going unanswered. A wedged robot leaves the
    // socket open and the keep-alive re-fires every second, so a level-logged
    // WARN would emit ~1/s and flush the whole ring in 20 seconds. Log the
    // transition in and the recovery out, never the steady state.
    bStateUnanswered : BOOL;

    // The same discipline, for connect failures. TRUE once an outage has been
    // reported, so the re-dial every ~3 s does not report it again.
    //
    // WHY THIS WAS NOT ALREADY HERE, and what it cost: bStateUnanswered got the
    // edge treatment in 2026-07-28 and the connect path never did, so with the
    // robot absent -- every bench session -- ALL 20 slots of GVL_Log.aRecent were
    // the same 'Connect failed' line at ~5 s spacing. The ring was fully
    // overwritten about every 100 seconds, which defeats this project's own rule
    // that transition paths must be read from GVL_Log rather than by polling
    // eStep. Phase 2 then made it worse by putting the same repeat on the Compact
    // Flash: the first CSV was 95% this one message, ~1.2 MB/day.
    bConnectFailed  : BOOL;

    // The error number that was reported. Guarding on the NUMBER as well as on the
    // boolean is the load-bearing part: a bare boolean would swallow a genuinely
    // NEW fault -- a wrong IP gives 1861 (timeout), a lost route gives something
    // else -- because the flag was already set by the first one. Silence about a
    // changed cause would be worse than the noise this removes.
    nLastConnectErr : UDINT;

    // Whether the in-flight TX should be traced at DBG. StartSend defaults it
    // TRUE for every frame; SendState overrides it to FALSE for a keep-alive
    // repeat, AFTER calling StartSend. Both halves are load-bearing: the
    // override must come second to win, and StartSend must clear it or a
    // keep-alive's FALSE would leak into the next real frame and hide it.
    bTraceTx : BOOL;
END_VAR
VAR
    // Endpoint actually dialled for the live session. sRemoteHost is only
    // read at connect time, so without this a commissioner who edits the IP
    // on the Robot page sees nothing happen until the socket happens to
    // drop -- the field would look broken.
    sDialledHost  : STRING;
    nDialledPort  : UINT;
    bDialledValid : BOOL;
END_VAR
VAR CONSTANT
    IO_IDLE      : INT := 0;
    IO_WAIT_SEND : INT := 1;
    IO_WAIT_RECV : INT := 2;

    PARAM_COUNT  : INT := 11;   // must match ST_RobotParams / SYNC_ORDER

    TX_NONE     : INT := 0;
    TX_GETSYNC  : INT := 1;
    TX_SETPARAM : INT := 2;
    TX_NEWBULB  : INT := 3;
    TX_STATE    : INT := 4;

    RECONNECT_MS   : TIME := T#3S;
    IDLE_STATE_MS  : TIME := T#1S;   // keep-alive STATE push cadence
    REPLY_TO_MS    : TIME := T#2S;
    CONNECT_TO_MS  : TIME := T#2S;
END_VAR

// Disable request routes an active session through the Error/close path.
// Logged at INFO, not ERR: an operator clearing bTcpEnable is not a fault.
IF NOT bEnable AND (eState = E_RobotConnState.Connecting OR eState = E_RobotConnState.Connected) THEN
    Fail(eSev := E_LogSev.INFO, sWhy := 'Disabled, closing link');
END_IF

// Endpoint retarget. The connect call reads sRemoteHost once, so a live
// session has to be torn down for a new IP to be dialled. Routed through
// Error, the same close-and-retry path the disable request uses, so the
// socket is released properly rather than leaked.
// Baselined on the first scan: without the guard the initial transition
// from an empty shadow would look like an edit and force a pointless
// reconnect at startup.
IF NOT bDialledValid THEN
    bDialledValid := TRUE;
    sDialledHost  := sRemoteHost;
    nDialledPort  := nRemotePort;
ELSIF (sRemoteHost <> sDialledHost) OR (nRemotePort <> nDialledPort) THEN
    sDialledHost := sRemoteHost;
    nDialledPort := nRemotePort;
    IF eState = E_RobotConnState.Connecting OR eState = E_RobotConnState.Connected THEN
        // INFO for the same reason as the disable path: a commissioner typing
        // a new IP is not a fault. Endpoint() already reads the NEW value --
        // sDialledHost was updated two lines up -- so the entry names where we
        // are going, which is the useful half.
        Fail(eSev := E_LogSev.INFO,
             sWhy := CONCAT('Endpoint changed, redialling ', Endpoint()));
    END_IF
END_IF

CASE eState OF

E_RobotConnState.Disconnected:
    tonReconnect(IN := TRUE, PT := RECONNECT_MS);
    IF bEnable AND tonReconnect.Q THEN
        tonReconnect(IN := FALSE);
        fbConnect(bExecute := FALSE);
        eState := E_RobotConnState.Connecting;
    END_IF

E_RobotConnState.Connecting:
    fbConnect(
        sSrvNetId   := sSrvNetId,
        sRemoteHost := sRemoteHost,
        nRemotePort := nRemotePort,
        bExecute    := TRUE,
        tTimeout    := CONNECT_TO_MS);
    IF NOT fbConnect.bBusy THEN
        fbConnect(bExecute := FALSE);
        IF fbConnect.bError THEN
            // The count is kept whatever we log, so a suppressed repeat is still
            // counted and visible on the Robot page.
            stRobot.nConnectFails := stRobot.nConnectFails + 1;

            // EDGE-GUARDED, exactly like bStateUnanswered. Report the first
            // failure of an outage at ERR, and report again whenever the error
            // NUMBER changes -- a new cause is new information and must get
            // through. A plain repeat of the same error is demoted to DBG, which
            // F_LogEvent drops unless GVL_Log.bDebugMode is set.
            //
            // DEMOTED RATHER THAN SUPPRESSED on purpose: ticking Debug still gives
            // the full retry trace when you actually want it, and the CSV writer
            // drops DBG unconditionally so the file never carries the repeat
            // either. nErrId is the whole diagnostic value here -- 'Connect
            // failed' alone cannot distinguish a wrong IP from a robot that is off.
            IF (NOT bConnectFailed) OR (fbConnect.nErrId <> nLastConnectErr) THEN
                bConnectFailed  := TRUE;
                nLastConnectErr := fbConnect.nErrId;
                Fail(eSev := E_LogSev.ERR,
                     sWhy := CONCAT(CONCAT('Connect failed ', Endpoint()),
                                    CONCAT(' err ', UDINT_TO_STRING(fbConnect.nErrId))));
            ELSE
                Fail(eSev := E_LogSev.DBG,
                     sWhy := CONCAT(CONCAT('Connect retry ', Endpoint()),
                                    CONCAT(' err ', UDINT_TO_STRING(fbConnect.nErrId))));
            END_IF
        ELSE
            hSocket         := fbConnect.hSocket;
            iIo             := IO_IDLE;
            iPend           := TX_NONE;
            nPendIdx        := 0;
            bAutoSyncQueued := TRUE;   // pull current params right after connect
            bShadowValid    := FALSE;  // no edit detection until that SYNC lands
            nLastStateSent  := -1;     // force initial STATE push
            tonIdle(IN := FALSE);

            // Reset the log edge-detectors with the rest of the session state,
            // so a reconnect re-reports an unanswered link or a repeated
            // command instead of staying quiet about it.
            bStateUnanswered := FALSE;
            nLastCmdLogged   := 0;

            eState := E_RobotConnState.Connected;

            // ONE INFO OUT, matching the one ERR in -- and it carries the count,
            // which is the point. 'Connected after 312 failed attempts' tells you
            // how long the outage lasted; 312 identical ERR lines do not, because
            // the ring only holds 20 of them and the oldest is what you needed.
            IF stRobot.nConnectFails > 0 THEN
                F_LogEvent(eSev := E_LogSev.INFO, sSource := stRobot.Name,
                           sMsg := CONCAT(CONCAT('Connected after ',
                                   CONCAT(UDINT_TO_STRING(stRobot.nConnectFails),
                                          ' failed attempts ')), Endpoint()));
            ELSE
                F_LogEvent(eSev := E_LogSev.INFO, sSource := stRobot.Name,
                           sMsg := CONCAT('Connected ', Endpoint()));
            END_IF

            // Re-arm the guard with the rest of the session state, so a LATER
            // outage reports again instead of staying quiet because an earlier
            // one had already set the flag.
            bConnectFailed        := FALSE;
            nLastConnectErr       := 0;
            stRobot.nConnectFails := 0;
        END_IF
    END_IF

E_RobotConnState.Connected:
    ConnectedIo();

E_RobotConnState.Error:
    fbClose(
        sSrvNetId := sSrvNetId,
        hSocket   := hSocket,
        bExecute  := TRUE,
        tTimeout  := CONNECT_TO_MS);
    IF NOT fbClose.bBusy THEN
        fbClose(bExecute := FALSE);
        MEMSET(ADR(hSocket), 0, SIZEOF(hSocket));
        iIo   := IO_IDLE;
        iPend := TX_NONE;
        tonReconnect(IN := FALSE);
        eState := E_RobotConnState.Disconnected;
    END_IF

END_CASE

// Mirror connection state to the HMI status struct.
stRobot.eConnState     := eState;
stRobot.sConnStateText := TO_STRING(eState);

// Request/reply sequencer, run while eState = Connected.
METHOD ConnectedIo : BOOL
VAR
    nChanged : INT;   // index of first param edited by the HMI, 0 = none
    nIdx     : INT;   // param index behind an explicit bSetParam name
    nRaw     : INT;   // value as the operator left it, before ClampParam
END_VAR
CASE iIo OF

IO_IDLE:
    tonIdle(IN := TRUE, PT := IDLE_STATE_MS);

    // Detect an operator edit: any of the 11 params differing from the
    // shadow snapshot taken after the last SYNC. Suppressed until the
    // first SYNC validates the shadow, otherwise the compiled-in defaults
    // would all look like edits on the very first scan after connect.
    IF bShadowValid THEN
        nChanged := FindChangedParam();
    ELSE
        nChanged := 0;
    END_IF

    // Priority order.
    //  1. The post-connect one-shot GET_SYNC, before anything else: the
    //     reply to a STATE push can carry CMD:1, and starting a cycle on
    //     parameters we have not read back yet would run the robot on
    //     stale values.
    //  2. A CHANGED state. CMD frames ride back on STATE replies, so
    //     delaying a state push behind a burst of parameter writes would
    //     also delay start/reset commands from the robot.
    //  3. Explicit requests, then detected edits.
    //  4. The keep-alive push last, where it only fires on an idle link.
    IF bAutoSyncQueued THEN
        bAutoSyncQueued := FALSE;
        sTxMsg := 'GET_SYNC';
        iPend  := TX_GETSYNC;
        StartSend();
    ELSIF stParams.nStateOut <> nLastStateSent THEN
        // A real state change: traced at DBG.
        SendState(bKeepAlive := FALSE);
    ELSIF stParams.bSetParam THEN
        // Explicit escape hatch: caller supplies the raw name/value pair.
        // Clamp it too, and write the clamped value back so the caller can
        // see what was actually sent. Unknown names pass through untouched --
        // that is the point of the escape hatch.
        nIdx := ParamIndex(stParams.sSetName);
        IF nIdx > 0 THEN
            nRaw             := stParams.nSetVal;
            stParams.nSetVal := ClampParam(i := nIdx, nVal := nRaw);
            IF stParams.nSetVal <> nRaw THEN
                LogClamp(i := nIdx, nRaw := nRaw, nSent := stParams.nSetVal);
            END_IF
        END_IF
        sTxMsg   := CONCAT(CONCAT(stParams.sSetName, ':'), INT_TO_STRING(stParams.nSetVal));
        iPend    := TX_SETPARAM;
        nPendIdx := 0;
        StartSend();
    ELSIF stParams.bTriggerNewBulb THEN
        sTxMsg := 'New_Bulb:1';
        iPend  := TX_NEWBULB;
        StartSend();
    ELSIF stParams.bGetSync THEN
        sTxMsg := 'GET_SYNC';
        iPend  := TX_GETSYNC;
        StartSend();
    ELSIF nChanged > 0 THEN
        // One param per round-trip; the next idle scan picks up the rest.
        //
        // Clamp, and write the clamped value BACK into the field before
        // sending. Writing back is not cosmetic: the shadow is updated to
        // the value we sent, so if the field kept the operator's
        // out-of-range number it would differ from the shadow forever and
        // the FB would re-send on every idle scan. Writing back converges,
        // and the HMI then shows what the robot actually got.
        nPendIdx := nChanged;
        nRaw     := ParamValue(nChanged);
        nPendVal := ClampParam(i := nChanged, nVal := nRaw);
        IF nPendVal <> nRaw THEN
            // Log BEFORE the write-back below overwrites the field: this is the
            // only moment the operator's original number still exists anywhere.
            LogClamp(i := nChanged, nRaw := nRaw, nSent := nPendVal);
        END_IF
        SetParamValue(i := nChanged, nVal := nPendVal);
        sTxMsg   := CONCAT(CONCAT(ParamName(nChanged), ':'), INT_TO_STRING(nPendVal));
        iPend    := TX_SETPARAM;
        StartSend();
    ELSIF tonIdle.Q THEN
        // Keep-alive repeat of a state already sent: deliberately not traced.
        SendState(bKeepAlive := TRUE);
    END_IF

IO_WAIT_SEND:
    fbSend(
        sSrvNetId := sSrvNetId,
        hSocket   := hSocket,
        cbLen     := TO_UDINT(LEN(sTxMsg)),
        pSrc      := ADR(sTxMsg),
        bExecute  := TRUE,
        tTimeout  := REPLY_TO_MS);
    IF NOT fbSend.bBusy THEN
        fbSend(bExecute := FALSE);
        IF fbSend.bError THEN
            Fail(eSev := E_LogSev.ERR,
                 sWhy := CONCAT(CONCAT('Send failed on ', PendName()),
                                CONCAT(' err ', UDINT_TO_STRING(fbSend.nErrId))));
        ELSE
            stRobot.nPacketsTx     := stRobot.nPacketsTx + 1;
            stRobot.sLastTxMessage := sTxMsg;
            // Traced here rather than in StartSend so the entry means "this
            // left the box", not "this was queued".
            IF bTraceTx THEN
                F_LogEvent(eSev := E_LogSev.DBG, sSource := stRobot.Name,
                           sMsg := CONCAT('TX ', LEFT(sTxMsg, 76)));
            END_IF
            tonReply(IN := FALSE);
            iIo := IO_WAIT_RECV;
        END_IF
    END_IF

IO_WAIT_RECV:
    tonReply(IN := TRUE, PT := REPLY_TO_MS);
    fbReceive(
        sSrvNetId := sSrvNetId,
        hSocket   := hSocket,
        cbLen     := SIZEOF(aRxBuffer) - 1,
        pDest     := ADR(aRxBuffer),
        bExecute  := TRUE,
        tTimeout  := REPLY_TO_MS);
    IF NOT fbReceive.bBusy THEN
        fbReceive(bExecute := FALSE);
        IF fbReceive.bError THEN
            Fail(eSev := E_LogSev.ERR,
                 sWhy := CONCAT(CONCAT('Recv failed on ', PendName()),
                                CONCAT(' err ', UDINT_TO_STRING(fbReceive.nErrId))));
        ELSIF fbReceive.nRecBytes > 0 THEN
            aRxBuffer[fbReceive.nRecBytes] := 0;   // null-terminate
            MEMCPY(ADR(sRxMsg), ADR(aRxBuffer), fbReceive.nRecBytes + 1);
            tonReply(IN := FALSE);
            HandleReply();
            iIo := IO_IDLE;
        ELSIF tonReply.Q THEN
            // No reply in time. STATE may go unanswered occasionally --
            // tolerate it (we'll try again next keep-alive); everything
            // else is a real fault -> drop and reconnect.
            tonReply(IN := FALSE);
            IF iPend = TX_STATE THEN
                // Edge-logged, not level-logged: the keep-alive re-fires every
                // second, so a WARN per unanswered push would flush the ring in
                // 20 entries and hide whatever caused it.
                IF NOT bStateUnanswered THEN
                    bStateUnanswered := TRUE;
                    F_LogEvent(eSev := E_LogSev.WARN, sSource := stRobot.Name,
                               sMsg := 'STATE unanswered, link may be stale');
                END_IF
                iPend := TX_NONE;
                iIo   := IO_IDLE;
            ELSE
                Fail(eSev := E_LogSev.ERR,
                     sWhy := CONCAT('Reply timeout on ', PendName()));
            END_IF
        END_IF
    END_IF

END_CASE
END_METHOD

// Arm a STATE:n push and remember what we sent.
METHOD SendState : BOOL
VAR_INPUT
    // TRUE when this is the 1 Hz keep-alive repeat of a state already sent.
    // Such frames are not traced at DBG -- at 1 Hz they would bury every other
    // entry in a 20-deep ring. Passed explicitly by the two call sites rather
    // than derived here, because deriving it would mean reading nLastStateSent
    // after the line below has already overwritten it.
    bKeepAlive : BOOL;
END_VAR
sTxMsg         := CONCAT('STATE:', INT_TO_STRING(stParams.nStateOut));
nLastStateSent := stParams.nStateOut;
iPend          := TX_STATE;
nPendIdx       := 0;
StartSend();

// Must come AFTER StartSend, which defaults bTraceTx TRUE for every frame.
bTraceTx := NOT bKeepAlive;
END_METHOD

// Index of the first param whose live value differs from the shadow
// snapshot, or 0 when everything matches.
METHOD FindChangedParam : INT
VAR
    i : INT;
END_VAR
FindChangedParam := 0;

FOR i := 1 TO PARAM_COUNT DO
    IF ParamValue(i) <> aShadow[i] THEN
        FindChangedParam := i;
        RETURN;
    END_IF
END_FOR
END_METHOD

// Re-baseline the shadow to the current stParams values and enable edit
// detection. Called after every GET_SYNC round-trip.
METHOD SetShadowAll : BOOL
VAR
    i : INT;
END_VAR
FOR i := 1 TO PARAM_COUNT DO
    aShadow[i] := ParamValue(i);
END_FOR

bShadowValid := TRUE;
END_METHOD

// Live value of param i. Index order must match ParamName and the
// robot's SYNC_ORDER.
METHOD ParamValue : INT
VAR_INPUT
    i : INT;
END_VAR
CASE i OF
     1: ParamValue := stParams.J_SPEED;
     2: ParamValue := stParams.L_SPEED;
     3: ParamValue := stParams.REPEATS;
     4: ParamValue := stParams.START_WAIT;
     5: ParamValue := stParams.WATER_WAIT;
     6: ParamValue := stParams.STAND_WAIT;
     7: ParamValue := stParams.END_WAIT;
     8: ParamValue := stParams.WATER_SPEED;
     9: ParamValue := stParams.WAX_WAIT_TIME_IN;
    10: ParamValue := stParams.WAX_WAIT_TIME_OUT;
    11: ParamValue := stParams.WAX_SPEED;
ELSE
    ParamValue := 0;
END_CASE
END_METHOD

// Write a value into param i. Inverse of ParamValue; same index order.
METHOD SetParamValue : BOOL
VAR_INPUT
    i    : INT;
    nVal : INT;
END_VAR
CASE i OF
     1: stParams.J_SPEED           := nVal;
     2: stParams.L_SPEED           := nVal;
     3: stParams.REPEATS           := nVal;
     4: stParams.START_WAIT        := nVal;
     5: stParams.WATER_WAIT        := nVal;
     6: stParams.STAND_WAIT        := nVal;
     7: stParams.END_WAIT          := nVal;
     8: stParams.WATER_SPEED       := nVal;
     9: stParams.WAX_WAIT_TIME_IN  := nVal;
    10: stParams.WAX_WAIT_TIME_OUT := nVal;
    11: stParams.WAX_SPEED         := nVal;
END_CASE
END_METHOD

// Index of a param by its wire name, or 0 if the name is not one of the
// eleven. Used to clamp the explicit bSetParam escape hatch; an unknown
// name deliberately returns 0 and is passed through unclamped.
METHOD ParamIndex : INT
VAR_INPUT
    sName : STRING(30);
END_VAR
VAR
    i : INT;
END_VAR
ParamIndex := 0;

FOR i := 1 TO PARAM_COUNT DO
    IF ParamName(i) = sName THEN
        ParamIndex := i;
        RETURN;
    END_IF
END_FOR
END_METHOD

(*
   Bound one parameter to the robot's documented range.

   These limits are the vendor's own: the Dobot-side tuning GUI
   (Robot\167-01-Saad\tcp client.py, PARAMS table + its clamp) refuses
   anything outside them, and readme.txt mirrors the same table. The robot's
   Lua (src2.lua) does NOT validate -- it assigns tonumber() straight
   through -- so nothing downstream of us catches a bad value.

   Clamping here rather than only on the VISU NumericInputs is deliberate:
   a per-control min/max bounds only that control, while every writer
   (panel, FlowerPyHmi over ADS, any future ADS client, and the bSetParam
   escape hatch) funnels through this FB.

   Units are percentages for the four speed values -- global.lua Init()
   passes J_SPEED / L_SPEED to VelJ() / VelL() and the WAX / WATER speeds to
   the v= velocity-ratio option of MovL. The waits are milliseconds.
*)
METHOD ClampParam : INT
VAR_INPUT
    i    : INT;
    nVal : INT;
END_VAR
ClampParam := LIMIT(ParamMin(i), nVal, ParamMax(i));
END_METHOD

// Lower bound of param i. Same index order as ParamValue / ParamName.
METHOD ParamMin : INT
VAR_INPUT
    i : INT;
END_VAR
CASE i OF
     1: ParamMin :=  1;    // J_SPEED            %
     2: ParamMin :=  1;    // L_SPEED            %
     3: ParamMin :=  1;    // REPEATS
     4: ParamMin := 10;    // START_WAIT         ms
     5: ParamMin := 10;    // WATER_WAIT         ms
     6: ParamMin := 10;    // STAND_WAIT         ms
     7: ParamMin := 10;    // END_WAIT           ms
     8: ParamMin :=  0;    // WATER_SPEED        %
     9: ParamMin :=  0;    // WAX_WAIT_TIME_IN   ms
    10: ParamMin := 10;    // WAX_WAIT_TIME_OUT  ms
    11: ParamMin :=  0;    // WAX_SPEED          %
ELSE
    ParamMin := 0;
END_CASE
END_METHOD

// Upper bound of param i. Same index order as ParamValue / ParamName.
METHOD ParamMax : INT
VAR_INPUT
    i : INT;
END_VAR
CASE i OF
     1: ParamMax :=   100;   // J_SPEED
     2: ParamMax :=   100;   // L_SPEED
     3: ParamMax :=    10;   // REPEATS
     4: ParamMax := 10000;   // START_WAIT
     5: ParamMax := 10000;   // WATER_WAIT
     6: ParamMax := 10000;   // STAND_WAIT
     7: ParamMax := 10000;   // END_WAIT
     8: ParamMax :=   100;   // WATER_SPEED
     9: ParamMax := 10000;   // WAX_WAIT_TIME_IN
    10: ParamMax := 10000;   // WAX_WAIT_TIME_OUT
    11: ParamMax :=   100;   // WAX_SPEED
ELSE
    ParamMax := 32767;
END_CASE
END_METHOD

// Wire name of param i, as the robot expects it in NAME:VALUE.
METHOD ParamName : STRING(30)
VAR_INPUT
    i : INT;
END_VAR
CASE i OF
     1: ParamName := 'J_SPEED';
     2: ParamName := 'L_SPEED';
     3: ParamName := 'REPEATS';
     4: ParamName := 'START_WAIT';
     5: ParamName := 'WATER_WAIT';
     6: ParamName := 'STAND_WAIT';
     7: ParamName := 'END_WAIT';
     8: ParamName := 'WATER_SPEED';
     9: ParamName := 'WAX_WAIT_TIME_IN';
    10: ParamName := 'WAX_WAIT_TIME_OUT';
    11: ParamName := 'WAX_SPEED';
ELSE
    ParamName := '';
END_CASE
END_METHOD

(*
   Log a reason and route the session into the Error state, which closes the
   socket and re-dials after RECONNECT_MS.

   Centralised so every teardown path is logged exactly once, by the code that
   knows why. Before this existed, six places assigned eState := Error and the
   HMI was left showing 'Disconnected' with no record of the cause.

   eSev is a parameter because two callers are NOT faults: an operator clearing
   bTcpEnable, and an endpoint retarget. Both reuse this same close-and-redial
   path deliberately, and logging either at ERR would cry wolf.
*)
METHOD Fail : BOOL
VAR_INPUT
    eSev : E_LogSev;
    sWhy : STRING(80);
END_VAR
F_LogEvent(eSev := eSev, sSource := stRobot.Name, sMsg := sWhy);
eState := E_RobotConnState.Error;
END_METHOD

// 'host:port' of the endpoint currently dialled, for log messages. Reads the
// dialled pair rather than the inputs, so an entry written during a retarget
// names what is actually being connected to.
METHOD Endpoint : STRING(60)
Endpoint := CONCAT(CONCAT(sDialledHost, ':'), UINT_TO_STRING(nDialledPort));
END_METHOD

// Wire name of the message awaiting a reply, so a send or timeout entry says
// WHICH exchange failed. 'Reply timeout' alone cannot distinguish a robot that
// never answers GET_SYNC from one that stopped mid-cycle.
METHOD PendName : STRING(20)
CASE iPend OF
    TX_GETSYNC:  PendName := 'GET_SYNC';
    TX_SETPARAM: PendName := 'SET';
    TX_NEWBULB:  PendName := 'New_Bulb';
    TX_STATE:    PendName := 'STATE';
ELSE
    PendName := 'none';
END_CASE
END_METHOD

// Report that a parameter write was bounded before it went out.
//
// WARN rather than INFO: the operator typed a number the robot would have
// taken literally, and ClampParam's write-back then replaces it in the field,
// so without this entry the edit appears to have simply not taken.
METHOD LogClamp : BOOL
VAR_INPUT
    i     : INT;   // param index
    nRaw  : INT;   // value as the operator left it
    nSent : INT;   // value actually transmitted
END_VAR
F_LogEvent(eSev := E_LogSev.WARN, sSource := stRobot.Name,
           sMsg := CONCAT(CONCAT(ParamName(i), ' '),
                          CONCAT(CONCAT(INT_TO_STRING(nRaw), ' out of range, clamped to '),
                                 INT_TO_STRING(nSent))));
END_METHOD

// Arm a send: reset edges/timers and enter the send wait state.
METHOD StartSend : BOOL
tonIdle(IN := FALSE);
fbSend(bExecute := FALSE);
iIo := IO_WAIT_SEND;

// Trace every frame by default. SendState is the only caller that opts out,
// and it does so after this returns. Clearing it here is what stops a
// keep-alive's opt-out from leaking into the next real frame.
bTraceTx := TRUE;
END_METHOD

// Dispatch on what we last sent; clear the consumed request flag.
METHOD HandleReply : BOOL
VAR
    bCmdSeen : BOOL;   // this reply carried a CMD: frame
    nCmd     : INT;    // its value, valid only when bCmdSeen
END_VAR
// Explicitly initialised rather than trusting method-local init: nCmd is only
// meaningful when bCmdSeen is TRUE, and every other method in this FB seeds its
// locals the same way. Seeded to -1, not 0, to match ParseCmd's "no CMD frame"
// return -- 0 would read as a genuine CMD:0 (withdraw command).
bCmdSeen := FALSE;
nCmd     := -1;

stRobot.nPacketsRx   := stRobot.nPacketsRx + 1;
stRobot.sLastMessage := sRxMsg;

// A reply of any kind proves the link is answering again.
IF bStateUnanswered THEN
    bStateUnanswered := FALSE;
    F_LogEvent(eSev := E_LogSev.INFO, sSource := stRobot.Name,
               sMsg := 'STATE replies resumed');
END_IF

// Any reply may embed the next robot command as "CMD:n". Parsed regardless of
// iPend so the state-push round-trip carries commands. ParseCmd returns -1 when
// the reply carries no CMD frame at all, which is what stops an 'OK: SET ...'
// ACK or a SYNC from clobbering a command still waiting for MAIN to consume it.
nCmd     := ParseCmd();
bCmdSeen := nCmd >= 0;

IF bCmdSeen THEN
    stParams.nRobotCmd := nCmd;
END_IF

// DBG frame trace. The idle 'CMD:0' answer to a keep-alive is the one reply
// deliberately not traced -- at 1 Hz it would bury everything else.
// LEFT bounds the string explicitly: a SYNC reply is longer than the 80 chars
// F_LogEvent takes, and an explicit truncation beats a silent one.
IF NOT (bCmdSeen AND nCmd = 0) THEN
    F_LogEvent(eSev := E_LogSev.DBG, sSource := stRobot.Name,
               sMsg := CONCAT('RX ', LEFT(sRxMsg, 76)));
END_IF

// Commands log on change. The robot may repeat one across several replies
// before zeroing it, and CMD:0 re-baselines without logging, so a genuine
// repeat of the same command after an intervening 0 still reports.
IF bCmdSeen AND (nCmd <> nLastCmdLogged) THEN
    nLastCmdLogged := nCmd;
    IF nCmd = 1 THEN
        F_LogEvent(eSev := E_LogSev.INFO, sSource := stRobot.Name,
                   sMsg := 'CMD:1 start cycle');
    ELSIF nCmd = 2 THEN
        F_LogEvent(eSev := E_LogSev.INFO, sSource := stRobot.Name,
                   sMsg := 'CMD:2 reset error');
    ELSIF nCmd <> 0 THEN
        // MAIN only acts on 1 and 2, so anything else is silently ignored
        // downstream. Worth a WARN rather than nothing at all.
        F_LogEvent(eSev := E_LogSev.WARN, sSource := stRobot.Name,
                   sMsg := CONCAT('CMD unknown, ignored: ', INT_TO_STRING(nCmd)));
    END_IF
END_IF

CASE iPend OF
    TX_GETSYNC:
        IF FIND(sRxMsg, 'SYNC:') = 1 THEN
            ParseSync();
            F_LogEvent(eSev := E_LogSev.INFO, sSource := stRobot.Name,
                       sMsg := 'SYNC ok, tuning params pulled');
        ELSE
            // SetShadowAll below deliberately runs anyway, so this WARN is the
            // only sign the pull produced nothing.
            F_LogEvent(eSev := E_LogSev.WARN, sSource := stRobot.Name,
                       sMsg := CONCAT('SYNC reply malformed: ', LEFT(sRxMsg, 54)));
        END_IF
        // Re-baseline unconditionally, even if the reply was malformed and
        // ParseSync did nothing. The shadow then equals whatever stParams
        // currently holds, so a pull never echoes straight back out as 11
        // spurious writes -- and the edit detector becomes live either way
        // instead of staying disabled behind one bad frame.
        SetShadowAll();
        stParams.bGetSync := FALSE;
    TX_SETPARAM:
        // Bank the value we actually sent, not the current field value: if
        // the operator edited the same param again mid-round-trip, the
        // mismatch survives and gets re-sent on the next idle scan.
        IF nPendIdx > 0 THEN
            // Logged before the shadow is banked -- aShadow still holds the
            // previous accepted value, which is the 'from' half of the entry.
            F_LogEvent(eSev := E_LogSev.INFO, sSource := stRobot.Name,
                       sMsg := CONCAT(CONCAT(ParamName(nPendIdx), ' '),
                                      CONCAT(CONCAT(INT_TO_STRING(aShadow[nPendIdx]), ' -> '),
                                             INT_TO_STRING(nPendVal))));
            aShadow[nPendIdx] := nPendVal;
            nPendIdx := 0;
        ELSE
            F_LogEvent(eSev := E_LogSev.INFO, sSource := stRobot.Name,
                       sMsg := CONCAT(CONCAT('SET ', stParams.sSetName),
                                      CONCAT(' = ', INT_TO_STRING(stParams.nSetVal))));
            stParams.bSetParam := FALSE;
        END_IF
    TX_NEWBULB:
        F_LogEvent(eSev := E_LogSev.INFO, sSource := stRobot.Name,
                   sMsg := 'New_Bulb acknowledged');
        stParams.bTriggerNewBulb := FALSE;
    TX_STATE:
        // CMD parsing already handled above; no flag to clear.
        ;
END_CASE

iPend := TX_NONE;
END_METHOD

(*
   Extract "CMD:<digit>" out of a reply and return its value, or -1 when the
   reply carries no usable CMD frame. -1 rather than 0 because 0 is itself a
   valid command (CMD:0 = withdraw), so the two cases must stay distinguishable:
   the caller only writes stParams.nRobotCmd when the result is >= 0, which is
   what stops a SYNC or an "OK: SET ..." ACK from clobbering a command that
   MAIN has not consumed yet.

   The write is left to the caller rather than done here so that it sits next
   to the logging that reports it -- HandleReply needs the value anyway to
   decide whether this command is a repeat worth suppressing.

   Deliberately more forgiving than the anchored one-liner it replaces
   (FIND(sRxMsg,'CMD:') = 1 plus MID over the tail), which required the
   frame to be EXACTLY 'CMD:' + digits:

   * Searches for the LAST occurrence rather than requiring position 1. The
     robot's Lua loop writes on a 100 ms tick while the PLC only reads once
     per round-trip, so two replies can coalesce into a single receive
     ('CMD:0CMD:1'). The old MID window then straddled the boundary and
     STRING_TO_INT returned 0 -- silently discarding a start request. Taking
     the last occurrence also means the newest command wins.
   * Reads exactly ONE digit and validates it, instead of assuming the digit
     is the final character. Trailing whitespace, a stray newline or any
     suffix the robot may append no longer parses as 0.

   m is single-digit by protocol (0=none, 1=start cycle, 2=reset error).
*)
METHOD ParseCmd : INT
VAR
    i     : INT;
    nLast : INT;   // 1-based position of the last 'CMD:' found, 0 = none
    nCh   : BYTE;
END_VAR
ParseCmd := -1;
nLast    := 0;

// Upper bound is LEN-4 so that both the 4-char tag and the digit that must
// follow it are inside the string. Shorter replies skip the loop entirely.
FOR i := 1 TO LEN(sRxMsg) - 4 DO
    IF MID(sRxMsg, 4, i) = 'CMD:' THEN
        nLast := i;
    END_IF
END_FOR

IF nLast > 0 THEN
    // String indexing is 0-based: 'CMD:' occupies nLast-1 .. nLast+2, so
    // the digit sits at nLast+3.
    nCh := sRxMsg[nLast + 3];
    IF nCh >= 16#30 AND nCh <= 16#39 THEN
        ParseCmd := TO_INT(nCh - 16#30);
    END_IF
END_IF
END_METHOD

// Parse "SYNC:NAME=VALUE,NAME=VALUE,..." into stParams.
METHOD ParseSync : BOOL
VAR
    sRest  : STRING(255);
    sToken : STRING(60);
    sName  : STRING(30);
    sVal   : STRING(20);
    nComma : INT;
    nEq    : INT;
    nLen   : INT;
    nGuard : INT;
END_VAR
nLen := LEN(sRxMsg);
IF nLen <= 5 THEN
    RETURN;
END_IF

// Strip the leading "SYNC:" (5 chars).
sRest := MID(sRxMsg, nLen - 5, 6);

nGuard := 0;
WHILE LEN(sRest) > 0 AND nGuard < 32 DO
    nGuard := nGuard + 1;

    nComma := FIND(sRest, ',');
    IF nComma > 0 THEN
        sToken := LEFT(sRest, nComma - 1);
        sRest  := MID(sRest, LEN(sRest) - nComma, nComma + 1);
    ELSE
        sToken := sRest;
        sRest  := '';
    END_IF

    nEq := FIND(sToken, '=');
    IF nEq > 0 THEN
        sName := LEFT(sToken, nEq - 1);
        sVal  := MID(sToken, LEN(sToken) - nEq, nEq + 1);
        ApplyParam(sName := sName, nVal := STRING_TO_INT(sVal));
    END_IF
END_WHILE
END_METHOD

// Assign one parsed NAME=VALUE pair into stParams.
METHOD ApplyParam : BOOL
VAR_INPUT
    sName : STRING(30);
    nVal  : INT;
END_VAR
IF    sName = 'J_SPEED'           THEN stParams.J_SPEED           := nVal;
ELSIF sName = 'L_SPEED'           THEN stParams.L_SPEED           := nVal;
ELSIF sName = 'REPEATS'           THEN stParams.REPEATS           := nVal;
ELSIF sName = 'START_WAIT'        THEN stParams.START_WAIT        := nVal;
ELSIF sName = 'WATER_WAIT'        THEN stParams.WATER_WAIT        := nVal;
ELSIF sName = 'STAND_WAIT'        THEN stParams.STAND_WAIT        := nVal;
ELSIF sName = 'END_WAIT'          THEN stParams.END_WAIT          := nVal;
ELSIF sName = 'WATER_SPEED'       THEN stParams.WATER_SPEED       := nVal;
ELSIF sName = 'WAX_WAIT_TIME_IN'  THEN stParams.WAX_WAIT_TIME_IN  := nVal;
ELSIF sName = 'WAX_WAIT_TIME_OUT' THEN stParams.WAX_WAIT_TIME_OUT := nVal;
ELSIF sName = 'WAX_SPEED'         THEN stParams.WAX_SPEED         := nVal;
END_IF
END_METHOD

END_FUNCTION_BLOCK

// ---- POUs/FB_PersistentAutoSave.TcPOU
(*
   Flushes the project's PERSISTENT config to disk a short while after the
   operator stops editing: all of GVL_HmiPersistent, plus GVL_Robot's
   commissioning endpoint (sRobotHost / nRobotPort).

   WHY THIS EXISTS. VAR_GLOBAL PERSISTENT declares a durable storage CLASS.
   It does not mean "saved automatically". TwinCAT writes RAM out to
   Port_851.bootdata on exactly three triggers: a clean PLC stop, an explicit
   FB_WritePersistentData call, or the IDE's PLC > Save persistent data menu.
   Cutting power to the CP6606 is not a clean stop, so before this FB existed
   every operator edit lived only in RAM and was silently lost on the next
   power cycle -- observed 2026-07-27 with tPlateWaitTimeoutMs reverting to
   its declared default.

   WHY DEBOUNCED. The panel boots from Compact Flash. Flushing on every
   keystroke would turn one edit of a 5-digit timeout into five writes. The
   FB waits for tQuietMs of no edits, so a burst collapses into one write.

   SAFETY NOTE. Making persistence work also makes the stMasterAutoCfg BOOLs
   survive a power cycle. MAIN's cold-boot block clears bContinuous on the
   first scan, because FB_MasterAutoCycle's IDLE branch tests it as a LEVEL
   and it is the one start path with no external gate -- restoring it TRUE
   would drive pistons within a scan of power-up. bAutoMode is deliberately
   NOT cleared (operator decision): the panel returns to Automatic and IDLE
   and still needs a real start trigger. Do not remove the cold-boot block
   without also removing this flush.
*)
FUNCTION_BLOCK FB_PersistentAutoSave
VAR_INPUT
    // Quiet period after the last edit before the flush fires.
    tQuietMs : UDINT := 2000;

    // AMS port of this PLC instance. 851 = first instance.
    nPort    : UINT  := 851;
END_VAR
VAR_OUTPUT
    bSaving    : BOOL;    // a flush is in progress
    bDirty     : BOOL;    // RAM differs from what we believe is on disk
    bError     : BOOL;    // last flush failed; see nErrorId
    nErrorId   : UDINT;   // ADS error from the last failed flush
    nSaveCount : UDINT;   // successful flushes since PLC start
END_VAR
VAR
    fbWrite    : Tc2_Utilities.FB_WritePersistentData;
    fbTrigDone : F_TRIG;   // falling edge of BUSY = the write finished
    tonQuiet   : TON;

    // Two shadow sets, which is what makes "stopped editing" detectable:
    //   shSaved = what we believe reached the disk. Refreshed only after a
    //             successful write, so bDirty means "a flush is owed".
    //   shSeen  = what we saw last scan. Refreshed every scan, so a
    //             difference means "changed during THIS scan".
    // The quiet timer runs only while dirty AND not changing, so it restarts
    // on every keystroke and elapses only once the operator stops.
    shSavedPiston : ARRAY[1..8] OF ST_HmiPistonAutoCfg;
    shSeenPiston  : ARRAY[1..8] OF ST_HmiPistonAutoCfg;
    shSavedMaster : ST_HmiMasterAutoCfg;
    shSeenMaster  : ST_HmiMasterAutoCfg;
    // Durable CSV log config (Phase 1 of docs/plans/log-csv-file.md). Without
    // these three edits -- declaration, baseline, compare -- stLogFileCfg is
    // PERSISTENT in storage class but never actually flushed, which is precisely
    // the defect this FB was written to fix.
    shSavedLogFile : ST_HmiLogFileCfg;
    shSeenLogFile  : ST_HmiLogFileCfg;

    // GVL_Robot's persistent commissioning endpoint. Lives in its own GVL
    // rather than GVL_HmiPersistent so its symbol paths stay stable, so it
    // has to be watched explicitly here. Scalars, so a plain <> works and
    // no MEMCMP is needed.
    shSavedHost : STRING;
    shSeenHost  : STRING;
    shSavedPort : UINT;
    shSeenPort  : UINT;

    // Bound once in section 0. An array of refs is the one case where a
    // POINTER beats VAR_IN_OUT here -- the alternative is eight near-identical
    // copies of the compare-and-baseline block.
    apPiston : ARRAY[1..8] OF POINTER TO ST_HmiPistonAutoCfg;

    bInit     : BOOL;
    bChanging : BOOL;
    bSaveReq  : BOOL;
    i         : INT;
END_VAR

(* ==========================================
   0. ONE-TIME BIND + BASELINE
   Baseline from the values ALREADY IN RAM, which at this point are the ones
   restored from bootdata. Baselining from the declared defaults instead
   would make every start look dirty and fire a pointless write.
   MAIN's cold-boot block runs before this FB is called, so the cleared
   The remaining cfg flags are part of the baseline and do not count as an
   edit either.
   ========================================== *)
IF NOT bInit THEN
    bInit := TRUE;
    apPiston[1] := ADR(GVL_HmiPersistent.stSepSol1AutoCfg);
    apPiston[2] := ADR(GVL_HmiPersistent.stSepSol2AutoCfg);
    apPiston[3] := ADR(GVL_HmiPersistent.stSepSol3AutoCfg);
    apPiston[4] := ADR(GVL_HmiPersistent.stPushSol1AutoCfg);
    apPiston[5] := ADR(GVL_HmiPersistent.stPushSol2AutoCfg);
    apPiston[6] := ADR(GVL_HmiPersistent.stPushSol3AutoCfg);
    apPiston[7] := ADR(GVL_HmiPersistent.stGripSolLAutoCfg);
    apPiston[8] := ADR(GVL_HmiPersistent.stGripSolRAutoCfg);

    FOR i := 1 TO 8 DO
        shSavedPiston[i] := apPiston[i]^;
        shSeenPiston[i]  := apPiston[i]^;
    END_FOR
    shSavedMaster := GVL_HmiPersistent.stMasterAutoCfg;
    shSeenMaster  := GVL_HmiPersistent.stMasterAutoCfg;

    shSavedLogFile := GVL_HmiPersistent.stLogFileCfg;
    shSeenLogFile  := GVL_HmiPersistent.stLogFileCfg;

    shSavedHost := GVL_Robot.sRobotHost;
    shSeenHost  := GVL_Robot.sRobotHost;
    shSavedPort := GVL_Robot.nRobotPort;
    shSeenPort  := GVL_Robot.nRobotPort;
END_IF

(* ==========================================
   1. CHANGE DETECTION
   MEMCMP rather than "<>" because IEC 61131-3 has no struct comparison.
   Padding bytes are compared too, but both sides are whole-struct copies of
   the same type, so padding matches and cannot cause a false positive.
   ========================================== *)
bDirty    := FALSE;
bChanging := FALSE;

FOR i := 1 TO 8 DO
    IF MEMCMP(apPiston[i], ADR(shSavedPiston[i]),
              SIZEOF(ST_HmiPistonAutoCfg)) <> 0 THEN
        bDirty := TRUE;
    END_IF
    IF MEMCMP(apPiston[i], ADR(shSeenPiston[i]),
              SIZEOF(ST_HmiPistonAutoCfg)) <> 0 THEN
        bChanging := TRUE;
        shSeenPiston[i] := apPiston[i]^;
    END_IF
END_FOR

IF MEMCMP(ADR(GVL_HmiPersistent.stMasterAutoCfg), ADR(shSavedMaster),
          SIZEOF(ST_HmiMasterAutoCfg)) <> 0 THEN
    bDirty := TRUE;
END_IF
IF MEMCMP(ADR(GVL_HmiPersistent.stMasterAutoCfg), ADR(shSeenMaster),
          SIZEOF(ST_HmiMasterAutoCfg)) <> 0 THEN
    bChanging := TRUE;
    shSeenMaster := GVL_HmiPersistent.stMasterAutoCfg;
END_IF

IF MEMCMP(ADR(GVL_HmiPersistent.stLogFileCfg), ADR(shSavedLogFile),
          SIZEOF(ST_HmiLogFileCfg)) <> 0 THEN
    bDirty := TRUE;
END_IF
IF MEMCMP(ADR(GVL_HmiPersistent.stLogFileCfg), ADR(shSeenLogFile),
          SIZEOF(ST_HmiLogFileCfg)) <> 0 THEN
    bChanging := TRUE;
    shSeenLogFile := GVL_HmiPersistent.stLogFileCfg;
END_IF

IF (GVL_Robot.sRobotHost <> shSavedHost)
OR (GVL_Robot.nRobotPort <> shSavedPort) THEN
    bDirty := TRUE;
END_IF
IF (GVL_Robot.sRobotHost <> shSeenHost)
OR (GVL_Robot.nRobotPort <> shSeenPort) THEN
    bChanging  := TRUE;
    shSeenHost := GVL_Robot.sRobotHost;
    shSeenPort := GVL_Robot.nRobotPort;
END_IF

(* ==========================================
   2. DEBOUNCE
   IN drops for the scan in which anything changed, resetting the timer. So
   Q fires only after tQuietMs with no edits at all, while still dirty.
   ========================================== *)
tonQuiet(IN  := bDirty AND NOT bChanging AND NOT fbWrite.BUSY,
         PT  := UDINT_TO_TIME(tQuietMs));

(* ==========================================
   3. FLUSH
   START is held high until BUSY rises so the request cannot be dropped if
   the ADS call has not been scheduled yet.
   ========================================== *)
IF tonQuiet.Q AND NOT fbWrite.BUSY THEN
    bSaveReq := TRUE;
END_IF

fbWrite(NETID := '', PORT := nPort, START := bSaveReq);
IF fbWrite.BUSY THEN
    bSaveReq := FALSE;
END_IF
bSaving := fbWrite.BUSY;

(* ==========================================
   4. COMPLETION
   Detected on the falling edge of BUSY rather than a DONE output, which
   FB_WritePersistentData does not expose.
   Re-baseline ONLY on success: after a failure the data is still owed to
   disk, so leaving shSaved alone keeps bDirty set and the FB retries once
   the operator's next edit settles.
   ========================================== *)
fbTrigDone(CLK := fbWrite.BUSY);

IF fbTrigDone.Q THEN
    IF fbWrite.ERR THEN
        bError   := TRUE;
        nErrorId := fbWrite.ERRID;
        F_LogEvent(eSev := E_LogSev.ERR, sSource := 'Persist',
                   sMsg := CONCAT('persistent save FAILED, ADS err ',
                                  UDINT_TO_STRING(fbWrite.ERRID)));
    ELSE
        bError   := FALSE;
        nErrorId := 0;
        FOR i := 1 TO 8 DO
            shSavedPiston[i] := apPiston[i]^;
        END_FOR
        shSavedMaster  := GVL_HmiPersistent.stMasterAutoCfg;
        // Refreshed ONLY here, on a successful write -- same as the others. If
        // this line were missing, stLogFileCfg would stay permanently different
        // from its saved shadow, bDirty would never clear, and the FB would
        // rewrite the whole persistent image every quiet period forever. On a
        // Compact Flash panel that is a wear bug, not just a wasted cycle.
        shSavedLogFile := GVL_HmiPersistent.stLogFileCfg;
        shSavedHost   := GVL_Robot.sRobotHost;
        shSavedPort   := GVL_Robot.nRobotPort;
        nSaveCount    := nSaveCount + 1;
        F_LogEvent(eSev := E_LogSev.INFO, sSource := 'Persist',
                   sMsg := 'persistent data saved');
    END_IF
END_IF

END_FUNCTION_BLOCK

// ---- POUs/FB_LogCsvWriter.TcPOU
(*
   Drains GVL_Log's 256-entry ring to a CSV file on the panel's Compact Flash.
   Phase 2 of docs/plans/log-csv-file.md. Called last in MAIN, after
   fbPersistentSave().

   WHY: the panel log is RAM only. Every entry is lost on power cycle, reset or
   download, so a fault overnight with nobody attached leaves nothing to read --
   which is exactly when the log matters most. This is the consumer the ring was
   designed for; its own comment has documented the drain contract
   (slot = nWriteIdx MOD 256) since long before anything drained it.

   Off by default. Nothing here touches the card until an operator sets
   GVL_HmiPersistent.stLogFileCfg.bEnabled.

   ---------------------------------------------------------------------------
   DELIBERATE DEVIATION FROM THE PLAN: no byte buffer.
   ---------------------------------------------------------------------------
   The plan says to accumulate rows into an ARRAY[0..2047] OF BYTE and flush it
   with one FB_FileWrite. This writes rows individually with FB_FilePuts inside a
   single open/close instead, for three reasons that only became clear once the
   Phase 0 probe had run on the real device:

     1. THE FLASH COST UNIT IS THE OPEN->CLOSE CYCLE, not the individual write.
        Data written between an open and a close reaches the OS cache and is
        committed once. So N Puts inside one open/close costs the card the same
        as one Write of N rows -- the flash economy the byte buffer existed for is
        preserved without the buffer.
     2. FB_FilePuts + FOPEN_MODETEXT IS THE ONLY FORM VERIFIED ON THIS TARGET.
        Measured 2026-08-10 by retrieving the probe's file over FTP: a single $N
        arrives as CRLF, exactly RFC 4180, and FilePuts adds no ending of its
        own. Whether text-mode translation also applies to FB_FileWrite's raw
        buffer is unverified -- and if it does, cbWriteLen no longer equals the
        bytes on disk and the size accounting silently drifts.
     3. THE RING IS ALREADY THE BUFFER. 256 entries of it. A second buffer would
        duplicate it and add a second place for entries to be lost.

   ---------------------------------------------------------------------------
   LINE ENDINGS: EVERY ROW ENDS WITH A BARE $N. NEVER $R$N.
   ---------------------------------------------------------------------------
   FOPEN_MODETEXT already turns LF into CRLF. Writing $R$N would have it
   translate the $N again, giving \r\r\n and a corrupt file. This was very nearly
   "fixed" the wrong way on the strength of a miscounted byte total; the measured
   file settled it. Do not change it without re-measuring.

   ---------------------------------------------------------------------------
   NEVER FALL BACK TO \Temp\ OR THE DEVICE ROOT \.
   ---------------------------------------------------------------------------
   Both are writable on this panel and BOTH LOSE THEIR CONTENTS ON RESTART -- the
   WinCE RAM object store. Proven 2026-08-10: files written there by the Phase 0
   probe were gone after an Activate, while the two on Compact Flash survived.
   A fallback to either would silently convert durable logging into RAM logging,
   reintroducing the exact defect this FB exists to fix, while every status field
   still reported healthy. A directory that cannot be opened must produce
   eState := FAILED with the error latched and visible. That is the whole point.
*)
FUNCTION_BLOCK FB_LogCsvWriter
VAR CONSTANT
    RING        : UDINT := 256;         // GVL_Log.aLog size -- the drain window
    HIGH_WATER  : UDINT := 200;         // flush early rather than risk overflow
    FILE_TO     : TIME  := T#5S;
    RETRY_TO    : TIME  := T#30S;       // backoff after a failure
    MAX_SKIP    : INT   := 32;          // DBG entries discarded per scan, bounded
    HDR         : STRING(40) := 'time,severity,source,message';
    E_NOTFOUND  : UDINT := 1804;        // ADS "file not found", verified on the panel
END_VAR
VAR
    eStep       : INT;

    fbMkDir     : Tc2_System.FB_CreateDir;
    fbProbe     : Tc2_System.FB_FileOpen;   // existence test, separate instance
    fbOpen      : Tc2_System.FB_FileOpen;
    fbPuts      : Tc2_System.FB_FilePuts;
    fbClose     : Tc2_System.FB_FileClose;
    hFile       : UINT;

    // Our own read cursor into the ring. The ONLY state that must not be lost
    // mid-session, and deliberately not persistent: after a reboot the ring is
    // empty and nWriteIdx restarts at 0, so a restored cursor would be ahead of
    // the writer and would skip everything until it caught up.
    udiLastRead : UDINT;
    bCursorSet  : BOOL;

    udiPending  : UDINT;
    sFileName   : STRING(40);
    sLastFile   : STRING(40);
    sPath       : STRING(160);
    sDirNoSlash : STRING(80);
    sRow        : STRING(255);
    nSlot       : INT;
    nSkipped    : INT;

    bNeedHeader : BOOL;
    bLossRow    : BOOL;         // a synthetic "entries lost" row is owed
    udiLostNow  : UDINT;
    bDirTried   : BOOL;
    bClosing    : BOOL;         // draining because bEnabled went FALSE
    bErrLogged  : BOOL;         // edge guard -- one ERR in, one INFO out

    tonFlush    : TON;
    tonRetry    : TON;
    fbTrigOff   : F_TRIG;
END_VAR

